// Reset FB
IF ( NOT Execute )
THEN
  Reset(); 
END_IF
END_METHOD

METHOD INTERNAL ParseResponsePayload : DINT
VAR_INPUT
  /// Response data
  ResponseData : RobotLibraryRecvDataFB;
  /// Timestamp
  Timestamp    : SystemTime;  
END_VAR
// TTable 6-172: Received CMD payload (RC to PLC) of "ReadLoadData"
// --------------------------
// Header
// --------------------------
// Byte 00 : USINT   - ParSeq | State     
// Byte 01 : SINT    - AlarmMessageSeverity    
// Byte 02 : UINT    - AlarmMessageCode HB
// Byte 03 :         - AlarmMessageCode LB
// --------------------------
// Datablock
// --------------------------
// Byte 04 : DATE    - LoadData.Date LW HB;
// Byte 05 :         - LoadData.Date LW LB;
// Byte 06 : TOD     - LoadData.Time LW HB;
// Byte 07 :         - LoadData.Time LW LB;
// Byte 08 :         - LoadData.Time LW HB;
// Byte 09 :         - LoadData.Time LW LB;
// Byte 10 : REAL    - LoadData.X HW HB;
// Byte 11 :         - LoadData.X HW LB;
// Byte 12 :         - LoadData.X LW HB;
// Byte 13 :         - LoadData.X LW LB;
// Byte 14 : REAL    - LoadData.Y HW HB;
// Byte 15 :         - LoadData.Y HW LB;
// Byte 16 :         - LoadData.Y LW HB;
// Byte 17 :         - LoadData.Y LW LB;
// Byte 18 : REAL    - LoadData.Z HW HB;
// Byte 19 :         - LoadData.Z HW LB;
// Byte 20 :         - LoadData.Z LW HB;
// Byte 21 :         - LoadData.Z LW LB;
// Byte 22 : REAL    - LoadData.RX HW HB;
// Byte 23 :         - LoadData.RX HW LB;
// Byte 24 :         - LoadData.RX LW HB;
// Byte 25 :         - LoadData.RX LW LB;
// Byte 26 : REAL    - LoadData.RY HW HB;
// Byte 27 :         - LoadData.RY HW LB;
// Byte 28 :         - LoadData.RY LW HB;
// Byte 29 :         - LoadData.RY LW LB;
// Byte 30 : REAL    - LoadData.RZ HW HB;
// Byte 31 :         - LoadData.RZ HW LB;
// Byte 32 :         - LoadData.RZ LW HB;
// Byte 33 :         - LoadData.RZ LW LB;
// Byte 34 : REAL    - LoadData.Mass HW HB;
// Byte 35 :         - LoadData.Mass HW LB;
// Byte 36 :         - LoadData.Mass LW HB;
// Byte 37 :         - LoadData.Mass LW LB;
// Byte 38 : REAL    - LoadData.IX HW HB;
// Byte 39 :         - LoadData.IX HW LB;
// Byte 40 :         - LoadData.IX LW HB;
// Byte 41 :         - LoadData.IX LW LB;
// Byte 42 : REAL    - LoadData.IY HW HB;
// Byte 43 :         - LoadData.IY HW LB;
// Byte 44 :         - LoadData.IY LW HB;
// Byte 45 :         - LoadData.IY LW LB;
// Byte 46 : REAL    - LoadData.IZ HW HB;
// Byte 47 :         - LoadData.IZ HW LB;
// Byte 48 :         - LoadData.IZ LW HB;
// Byte 49 :         - LoadData.IZ LW LB;
// Byte 50 : USINT   - LoadNo;
// Byte 51 : BOOL    - DataChanged;
// --------------------------
// call base implementation to parse the header from payload buffer
ResponseData.PayloadPtr := SUPER^.ParseResponsePayload(ResponseData := ResponseData, Timestamp := Timestamp);

// copy parsed header to response
_response.ParSeq               := _rspHeader.ParSeq;
_response.State                := _rspHeader.State;
_response.AlarmMessageSeverity := _rspHeader.AlarmMessageSeverity;
_response.AlarmMessageCode     := _rspHeader.AlarmMessageCode;

// Get Response.LoadData.Timestamp.IEC_DATE
_response.LoadData.Timestamp.IEC_DATE := ResponseData.GetIecDate();
// Get Response.LoadData.Timestamp.IEC_TIME
_response.LoadData.Timestamp.IEC_TIME := ResponseData.GetIecTime();
// Get Response.LoadData.X
_response.LoadData.X := ResponseData.GetReal();
// Get Response.LoadData.Y
_response.LoadData.Y := ResponseData.GetReal();
// Get Response.LoadData.Z
_response.LoadData.Z := ResponseData.GetReal();
// Get Response.LoadData.Rx
_response.LoadData.Rx := ResponseData.GetReal();
// Get Response.LoadData.Ry
_response.LoadData.Ry := ResponseData.GetReal();
// Get Response.LoadData.Rz
_response.LoadData.Rz := ResponseData.GetReal();
// Get Response.LoadData.Mass
_response.LoadData.Mass := ResponseData.GetReal();
// Get Response.LoadData.Ix
_response.LoadData.Ix := ResponseData.GetReal();
// Get Response.LoadData.Iy
_response.LoadData.Iy := ResponseData.GetReal();
// Get Response.LoadData.Iz
_response.LoadData.Iz := ResponseData.GetReal();
// Get Response.LoadNoReturn
_response.LoadNoReturn := ResponseData.GetUsint();
// Get Response.DataChanged
_response.DataChanged := ResponseData.GetBool();

// Create logging
ParseResponsePayloadLog(ResponseData := ResponseData, Timestamp := Timestamp);
END_METHOD

METHOD INTERNAL ParseResponsePayloadLog
VAR_INPUT
  /// Response data
  ResponseData : RobotLibraryRecvDataFB;
  /// Timestamp
  Timestamp    : SystemTime;  
END_VAR
// Create log entry for Parameter start
CreateLogMessage      ( Timestamp   := Timestamp,
                        MessageType := MessageType.CMD,
                        Severity    := Severity.DEBUG,
                        MessageCode := 0,
                        MessageText := 'Parsed the following parameter(s) from response data:');

// Create log entry for LoadData.Timestamp.IEC_DATE
CreateLogMessagePara1 ( Timestamp   := Timestamp,
                        MessageType := MessageType.CMD,
                        Severity    := Severity.DEBUG,
                        MessageCode := 0,
                        MessageText := 'Response.LoadData.Timestamp.IEC_DATE = {1}',
                        Para1       :=  IEC_DATE_TO_STRING(_response.LoadData.Timestamp.IEC_DATE));

// Create log entry for LoadData.Timestamp.IEC_TIME
CreateLogMessagePara1 ( Timestamp   := Timestamp,
                        MessageType := MessageType.CMD,
                        Severity    := Severity.DEBUG,
                        MessageCode := 0,
                        MessageText := 'Response.LoadData.Timestamp.IEC_TIME = {1}',
                        Para1       :=  IEC_TIME_TO_STRING(_response.LoadData.Timestamp.IEC_TIME));
                        
// Create log entry for LoadData.X
CreateLogMessagePara1 ( Timestamp   := Timestamp,
                        MessageType := MessageType.CMD,
                        Severity    := Severity.DEBUG,
                        MessageCode := 0,
                        MessageText := 'Response.LoadData.X = {1}',
                        Para1       :=  REAL_TO_STRING(_response.LoadData.X));

// Create log entry for LoadData.Y
CreateLogMessagePara1 ( Timestamp   := Timestamp,
                        MessageType := MessageType.CMD,
                        Severity    := Severity.DEBUG,
                        MessageCode := 0,
                        MessageText := 'Response.LoadData.Y = {1}',
                        Para1       :=  REAL_TO_STRING(_response.LoadData.Y));

// Create log entry for LoadData.Z
CreateLogMessagePara1 ( Timestamp   := Timestamp,
                        MessageType := MessageType.CMD,
                        Severity    := Severity.DEBUG,
                        MessageCode := 0,
                        MessageText := 'Response.LoadData.Z = {1}',
                        Para1       :=  REAL_TO_STRING(_response.LoadData.Z));

// Create log entry for LoadData.Rx
CreateLogMessagePara1 ( Timestamp   := Timestamp,
                        MessageType := MessageType.CMD,
                        Severity    := Severity.DEBUG,
                        MessageCode := 0,
                        MessageText := 'Response.LoadData.Rx = {1}',
                        Para1       :=  REAL_TO_STRING(_response.LoadData.Rx));

// Create log entry for LoadData.Ry
CreateLogMessagePara1 ( Timestamp   := Timestamp,
                        MessageType := MessageType.CMD,
                        Severity    := Severity.DEBUG,
                        MessageCode := 0,
                        MessageText := 'Response.LoadData.Ry = {1}',
                        Para1       :=  REAL_TO_STRING(_response.LoadData.Ry));

// Create log entry for LoadData.Rz
CreateLogMessagePara1 ( Timestamp   := Timestamp,
                        MessageType := MessageType.CMD,
                        Severity    := Severity.DEBUG,
                        MessageCode := 0,
                        MessageText := 'Response.LoadData.Rz = {1}',
                        Para1       :=  REAL_TO_STRING(_response.LoadData.Rz));

// Create log entry for LoadData.Mass
CreateLogMessagePara1 ( Timestamp   := Timestamp,
                        MessageType := MessageType.CMD,
                        Severity    := Severity.DEBUG,
                        MessageCode := 0,
                        MessageText := 'Response.LoadData.Mass = {1}',
                        Para1       :=  REAL_TO_STRING(_response.LoadData.Mass));

// Create log entry for LoadData.Ix
CreateLogMessagePara1 ( Timestamp   := Timestamp,
                        MessageType := MessageType.CMD,
                        Severity    := Severity.DEBUG,
                        MessageCode := 0,
                        MessageText := 'Response.LoadData.Ix = {1}',
                        Para1       :=  REAL_TO_STRING(_response.LoadData.Ix));

// Create log entry for LoadData.Iz
CreateLogMessagePara1 ( Timestamp   := Timestamp,
                        MessageType := MessageType.CMD,
                        Severity    := Severity.DEBUG,
                        MessageCode := 0,
                        MessageText := 'Response.LoadData.Iz = {1}',
                        Para1       :=  REAL_TO_STRING(_response.LoadData.Iz));

// Create log entry for LoadData.Iy
CreateLogMessagePara1 ( Timestamp   := Timestamp,
                        MessageType := MessageType.CMD,
                        Severity    := Severity.DEBUG,
                        MessageCode := 0,
                        MessageText := 'Response.LoadData.Iy = {1}',
                        Para1       :=  REAL_TO_STRING(_response.LoadData.Iy));

  // Create log entry for LoadNoReturn
CreateLogMessagePara1 ( Timestamp   := Timestamp,
                        MessageType := MessageType.CMD,
                        Severity    := Severity.DEBUG,
                        MessageCode := 0,
                        MessageText := 'Response.LoadNoReturn = {1}',
                        Para1       :=  USINT_TO_STRING(_response.LoadNoReturn));

  // Create log entry for DataChanged
CreateLogMessagePara1 ( Timestamp   := Timestamp,
                        MessageType := MessageType.CMD,
                        Severity    := Severity.DEBUG,
                        MessageCode := 0,
                        MessageText := 'Response.DataChanged = {1}',
                        Para1       :=  BOOL_TO_STRING(_response.DataChanged));
END_METHOD

METHOD PROTECTED Reset : DINT
VAR_INPUT
END_VAR
Reset := SUPER^.Reset();

Done               := FALSE;
Busy               := FALSE;
CommandBuffered    := FALSE;
END_METHOD

END_FUNCTION_BLOCK

// Library/POUs/Read/MC_ReadReals/MC_ReadRealsFB
/// Read real values on RC
FUNCTION_BLOCK MC_ReadRealsFB EXTENDS RobotLibraryBaseExecuteFB
// ------------------------------------------------------------------------- 
//  SRCI Robot Library                                                
// ------------------------------------------------------------------------- 
//                                                                           
//  Object:      ReadRealsFB                                       
//  Author:      Thorsten Brach                                                
//  Date:        2024-06-01
//
//  Description:                                              
//   
//                                                                           
//  Copyright: 
//    (C) 2024 Thorsten Brach. All rights reserved                                                                                                                                            
//             Licensed under the LGPL-3.0 license.
//                                                                           
//  Disclaimer:                                                                           
//    This project is provided without any guarantee and can be used for   
//    private and commercial purposes. Any use is at the user’s 
//    own risk and responsibility.
//
// -------------------------------------------------------------------------
VAR_INPUT
  /// Processing Mode
  ProcessingMode     : ProcessingMode;
  /// Defines the target sequence in which the command will be executed
  SequenceFlag       : SequenceFlag;
  /// command parameter 
  ParCmd             : ReadRealsParCmd;
END_VAR
VAR_OUTPUT
  /// TRUE, while the following outputs return valid values:
  /// • Values
  Valid              : BOOL; 
  /// Command is transferred and confirmed by the RC
  CommandBuffered    : BOOL;
  /// The command was aborted by another command.
  CommandAborted     : BOOL;
  /// TRUE, while command is interrupted during execution and can be continued
  CommandInterrupted : BOOL;
  /// command outputs
  OutCmd             : ReadRealsOutCmd;       
END_VAR

VAR
  /// internal copy of command parameter 
 _parCmd             : ReadRealsParCmd;
  /// command data to send
 _command            : ReadRealsSendData;
  /// response data received
 _response           : ReadRealsRecvData;      
END_VAR

SUPER^(AxesGroup := AxesGroup);

METHOD PROTECTED CheckFunctionSupported : BOOL
VAR_IN_OUT
  /// Robot assignment of function
  AxesGroup : AxesGroup; 
END_VAR
CheckFunctionSupported := AxesGroup.InternalData.RCSupportedFunctions.ReadReals;

IF ( NOT CheckFunctionSupported )
THEN
  // call base implementation for set error and create log entry
  SUPER^.CheckFunctionSupported(AxesGroup := AxesGroup);
END_IF
END_METHOD

METHOD PROTECTED CheckParameterChanged : BOOL
VAR_IN_OUT
  /// Robot assignment of function
  AxesGroup    : AxesGroup; 
END_VAR
// Check ParCmd Size is > 0, because MemCmp does not work correctly with size = 0
IF (SIZEOF(ParCmd) = 0) 
THEN 
  RETURN;
END_IF

// compare memory 
_parameterChanged := ( SysDepMemCmp(pData1 := ADR(ParCmd), pData2 := ADR(_parCmd), DataLen := SIZEOF(ParCmd)) <> RobotLibraryConstants.OK );

// check parameter valid ?
_parameterValid   := CheckParameterValid( AxesGroup := AxesGroup );

IF ((  _parameterChanged        )  AND 
    (  _parameterValid          )) OR
    (  _parameterUpdateInternal )  
THEN  
  // reset internal flag for send parameter update
 _parameterUpdateInternal := FALSE;
  // update internal copy of parameters 
 _parCmd := ParCmd;
  // inc parameter sequence
 _command.ParSeq := _command.ParSeq + 1;
  // update command data  
  CommandData := CreateCommandPayload(AxesGroup := AxesGroup); // ( Access via reference to rCommandFB in ACR )
  // notify active command register 
  AxesGroup.Acyclic.ActiveCommandRegister.NotifyParameterChanged := _uniqueID;
END_IF
END_METHOD

METHOD INTERNAL CreateCommandPayload : RobotLibrarySendDataFB
VAR_IN_OUT
  /// Robot assignment of function
  AxesGroup : AxesGroup; 
END_VAR
// Table 6-502: Sent CMD payload (PLC to RC) of "ReadReals"
// --------------------------
// Header
// --------------------------
// Byte 00 : UINT  - Type HB     
// Byte 01 :       - Type LB    
// Byte 02 : USINT - Reserve | ExecutionMode
// Byte 03 : USINT - ParSeq  | Priority
// --------------------------
// Datablock
// --------------------------
// Byte 04 : SINT  EmitterID[0];
// Byte 05 : SINT  EmitterID[1];
// Byte 06 : SINT  EmitterID[2];
// Byte 07 : SINT  EmitterID[3];
// Byte 08 : SINT  ListenerID;
// Byte 09 : BYTE  Reserved;
// Byte 10 : USINT Index[0];
// Byte 11 : USINT Index[1];
// Byte 12 : USINT Index[2];
// Byte 13 : USINT Index[3];
// Byte 14 : USINT Index[4];
// Byte 14 : USINT Index[5];
// Byte 14 : USINT Index[6];
// --------------------------
// set command parameter 
_command.CmdTyp       :=  CmdType.ReadReals;
_command.ExecMode     :=  ExecMode;
_command.ParSeq       := _command.ParSeq;
_command.Priority     :=  Priority;
_command.EmitterID[0] := 0;
_command.EmitterID[1] := 0;
_command.EmitterID[2] := 0;
_command.EmitterID[3] := 0;
_command.Reserve      := 0;
_command.ListenerID   := _parCmd.ListenerID;
_command.Index        := _parCmd.Index;


// copy command data to header
_cmdHeader := _command;
// call base implementation to copy header to payload buffer
CreateCommandPayload := SUPER^.CreateCommandPayload(AxesGroup := AxesGroup);

// add command.EmitterID[0]
CreateCommandPayload.AddSint(_command.EmitterID[0]);
// add command.EmitterID[1]
CreateCommandPayload.AddSint(_command.EmitterID[1]);
// add command.EmitterID[2]
CreateCommandPayload.AddSint(_command.EmitterID[2]);
// add command.EmitterID[3]
CreateCommandPayload.AddSint(_command.EmitterID[3]);
// add command.ListenerID
CreateCommandPayload.AddSint(_command.ListenerID);
// add command.Reserve
CreateCommandPayload.AddSint(_command.Reserve);
// add command.Index[0]
CreateCommandPayload.AddUsint(_command.Index[0]);
// add command.Index[1]
CreateCommandPayload.AddUsint(_command.Index[1]);
// add command.Index[2]
CreateCommandPayload.AddUsint(_command.Index[2]);
// add command.Index[3]
CreateCommandPayload.AddUsint(_command.Index[3]);
// add command.Index[4]
CreateCommandPayload.AddUsint(_command.Index[4]);
// add command.Index[5]
CreateCommandPayload.AddUsint(_command.Index[5]);
// add command.Index[6]
CreateCommandPayload.AddUsint(_command.Index[6]);

// Create logging
CreateCommandPayloadLog(AxesGroup := AxesGroup);
END_METHOD

METHOD INTERNAL CreateCommandPayloadLog
VAR_IN_OUT
  /// Robot assignment of function
  AxesGroup : AxesGroup; 
END_VAR
VAR 
  /// internal index for loops
 _idx : DINT;
END_VAR
// Create log entry for Parameter start
CreateLogMessage      ( Timestamp   := AxesGroup.InternalData.SystemTime,
                        MessageType := MessageType.CMD,
                        Severity    := Severity.DEBUG,
                        MessageCode := 0,
                        MessageText := 'Create command payload with the following parameter(s) :');
  
// Create log entry for EmitterID[x]
FOR _idx := 0 TO 3
DO
  CreateLogMessagePara2 ( Timestamp   := AxesGroup.InternalData.SystemTime,
                          MessageType := MessageType.CMD,
                          Severity    := Severity.DEBUG,
                          MessageCode := 0,
                          MessageText := 'Command.EmitterID[{2}] = {1}',
                          Para1       :=  SINT_TO_STRING(_command.EmitterID[_idx]),
                          Para2       :=  DINT_TO_STRING(_idx));
END_FOR

// Create log entry for ListenerID
CreateLogMessagePara1 ( Timestamp   := AxesGroup.InternalData.SystemTime,
                        MessageType := MessageType.CMD,
                        Severity    := Severity.DEBUG,
                        MessageCode := 0,
                        MessageText := 'Command.ListenerID = {1}',
                        Para1       :=  SINT_TO_STRING(_command.ListenerID));
                        
// Create log entry for Reserve
CreateLogMessagePara1 ( Timestamp   := AxesGroup.InternalData.SystemTime,
                        MessageType := MessageType.CMD,
                        Severity    := Severity.DEBUG,
                        MessageCode := 0,
                        MessageText := 'Command.Reserve = {1}',
                        Para1       :=  SINT_TO_STRING(_command.Reserve));

// Create log entry for Index[x]
FOR _idx := 0 TO 6
DO
  CreateLogMessagePara2 ( Timestamp   := AxesGroup.InternalData.SystemTime,
                          MessageType := MessageType.CMD,
                          Severity    := Severity.DEBUG,
                          MessageCode := 0,
                          MessageText := 'Command.Index[{2}] = {1}',
                          Para1       :=  USINT_TO_STRING(_command.Index[_idx]),
                          Para2       :=  DINT_TO_STRING(_idx));
END_FOR
END_METHOD

METHOD FB_init : BOOL
VAR_INPUT
  /// if TRUE, the retain variables are initialized (warm start / cold start)
  bInitRetains : BOOL; 
  /// if TRUE, the instance afterwards gets moved into the copy code (online change)
  bInCopyCode  : BOOL;  
END_VAR
MyType := 'MC_ReadRealsFB';

ExecMode := ExecutionMode.PARALLEL;
END_METHOD

METHOD PROTECTED OnCall
VAR_IN_OUT
  /// Robot assignment of function
  AxesGroup : AxesGroup; 
END_VAR
// call base implementation
SUPER^.OnCall(AxesGroup := AxesGroup);

CASE _stepCmd OF
  
  00:  IF ( _execute_R.Q )  
       THEN
         // Check function is supported and parameter are valid ?
         IF (( CheckFunctionSupported( AxesGroup := AxesGroup )) AND
             ( CheckParameterValid   ( AxesGroup := AxesGroup )))
         THEN      
           // set busy flag
           Busy := TRUE;
           // Reset command outputs
           SysDepMemSet(pDest := ADR(OutCmd), Value := 0, DataLen := SIZEOF(OutCmd));         
           // apply command parameter
          _parCmd := ParCmd;
           // init parameter sequence
          _command.ParSeq := 1;
           // create command data
           CommandData := CreateCommandPayload(AxesGroup := AxesGroup);
           // Add command to active command register
          _uniqueID := AxesGroup.Acyclic.ActiveCommandRegister.AddCmd( pCommandFB := ADR(THIS^ ));     
           // set timeout
           SetTimeout(PT := _timeoutCmd, rTimer := _timerCmd);
           // inc step counter
          _stepCmd := _stepCmd + 1;
         END_IF 
       END_IF
     

  01:  // Wait for responce received
       IF ( _responseReceived )
       THEN
         // reset response received flag
        _responseReceived := FALSE;

         CASE  _response.State 
         OF
           CmdMessageState.BUFFERED    : CommandBuffered    := TRUE;
           CmdMessageState.INTERRUPTED : CommandInterrupted := TRUE;           
           CmdMessageState.DONE        : Done               := TRUE;           
           CmdMessageState.ABORTED     : CommandAborted     := TRUE;
           CmdMessageState.ERROR       : Error              := TRUE;
         END_CASE
                
         // Done, Aborted or Error ?
         IF (_response.State >= CmdMessageState.DONE )
         THEN
           // Reset Busy flag
           Busy := FALSE;
           // Update results
           OutCmd.OriginID          := _response.OriginID;
           OutCmd.InvocationCounter := _response.InvocationCounter;
           OutCmd.Values            := _response.Values;
           
           // set timeout
           SetTimeout(PT := _timeoutCmd, rTimer := _timerCmd);
           // inc step counter
          _stepCmd := _stepCmd + 1; 
         END_IF
       END_IF


  02: IF ( NOT Execute)
      THEN
        Reset();
      END_IF
     
ELSE
  // invalid step
  ErrorID := RobotLibraryEvents.ERR_INVALID_STEP;
END_CASE


// Reset FB
IF ( NOT Execute )
THEN
  Reset();
END_IF
END_METHOD

METHOD INTERNAL ParseResponsePayload : DINT
VAR_INPUT
  /// Response data
  ResponseData : RobotLibraryRecvDataFB;
  /// Timestamp
  Timestamp    : SystemTime;  
END_VAR
VAR 
  /// internal index for loops
 _idx : DINT;
END_VAR
// Table Table 6-503: Received CMD payload (RC to PLC) of "ReadReals"
// --------------------------
// Header
// --------------------------
// Byte 00 : USINT   - ParSeq | State     
// Byte 01 : SINT    - AlarmMessageSeverity    
// Byte 02 : UINT    - AlarmMessageCode HB
// Byte 03 :         - AlarmMessageCode LB
// --------------------------
// Datablock
// --------------------------
// Byte 04 : USINT   - InvocationCounter;
// Byte 05 : SINT    - Reserved;
// Byte 06 : INT     - OriginID HW HB;
// Byte 07 :         - OriginID HW LB;
// Byte 08 : REAL    - Values[0] HW HB;
// Byte 09 :         - Values[0] HW LB;
// Byte 10 :         - Values[0] LW HB;
// Byte 11 :         - Values[0] LW LB;
// Byte 12 : REAL    - Values[1] HW HB;
// Byte 13 :         - Values[1] HW LB;
// Byte 14 :         - Values[1] LW HB;
// Byte 15 :         - Values[1] LW LB;
// Byte 16 : REAL    - Values[2] HW HB;
// Byte 17 :         - Values[2] HW LB;
// Byte 18 :         - Values[2] LW HB;
// Byte 19 :         - Values[2] LW LB;
// Byte 20 : REAL    - Values[3] HW HB;
// Byte 21 :         - Values[3] HW LB;
// Byte 22 :         - Values[3] LW HB;
// Byte 23 :         - Values[3] LW LB;
// Byte 24 : REAL    - Values[4] HW HB;
// Byte 25 :         - Values[4] HW LB;
// Byte 26 :         - Values[4] LW HB;
// Byte 27 :         - Values[4] LW LB;
// Byte 28 : REAL    - Values[5] HW HB;
// Byte 29 :         - Values[5] HW LB;
// Byte 30 :         - Values[5] LW HB;
// Byte 31 :         - Values[5] LW LB;
// Byte 32 : REAL    - Values[6] HW HB;
// Byte 33 :         - Values[6] HW LB;
// Byte 34 :         - Values[6] LW HB;
// Byte 35 :         - Values[6] LW LB;
// --------------------------
// call base implementation to parse the header from payload buffer
ResponseData.PayloadPtr := SUPER^.ParseResponsePayload(ResponseData := ResponseData, Timestamp := Timestamp);

// copy parsed header to response
_response.ParSeq               := _rspHeader.ParSeq;
_response.State                := _rspHeader.State;
_response.AlarmMessageSeverity := _rspHeader.AlarmMessageSeverity;
_response.AlarmMessageCode     := _rspHeader.AlarmMessageCode;

// Get Response.InvocationCounter
_response.InvocationCounter := ResponseData.GetUsint();
// Get Response.Reserve
_response.Reserve := ResponseData.GetSint();
// Get Response.OriginID/
_response.OriginID := ResponseData.GetInt();

// Get Response.Values[0]
FOR _idx := 0 TO 6 
DO
 _response.Values[_idx] := ResponseData.GetReal();
END_FOR

// Create logging
ParseResponsePayloadLog(ResponseData := ResponseData, Timestamp := Timestamp);
END_METHOD

METHOD INTERNAL ParseResponsePayloadLog
VAR_INPUT
  /// Response data
  ResponseData : RobotLibraryRecvDataFB;
  /// Timestamp
  Timestamp    : SystemTime;  
END_VAR
VAR 
  /// internal index for loops
 _idx : DINT;
END_VAR
// Create log entry for Parameter start
CreateLogMessage      ( Timestamp   := Timestamp,
                        MessageType := MessageType.CMD,
                        Severity    := Severity.DEBUG,
                        MessageCode := 0,
                        MessageText := 'Parsed the following parameter(s) from response data:');
                        
// Create log entry for InvocationCounter
CreateLogMessagePara1 ( Timestamp   := Timestamp,
                        MessageType := MessageType.CMD,
                        Severity    := Severity.DEBUG,
                        MessageCode := 0,
                        MessageText := 'Response.InvocationCounter = {1}',
                        Para1       :=  USINT_TO_STRING(_response.InvocationCounter));

// Create log entry for Reserve
CreateLogMessagePara1 ( Timestamp   := Timestamp,
                        MessageType := MessageType.CMD,
                        Severity    := Severity.DEBUG,
                        MessageCode := 0,
                        MessageText := 'Response.Reserve = {1}',
                        Para1       :=  SINT_TO_STRING(_response.Reserve));

// Create log entry for OriginID
CreateLogMessagePara1 ( Timestamp   := Timestamp,
                        MessageType := MessageType.CMD,
                        Severity    := Severity.DEBUG,
                        MessageCode := 0,
                        MessageText := 'Response.OriginID = {1}',
                        Para1       :=  INT_TO_STRING(_response.OriginID));

// Create log entry for Values[{x}]
FOR _idx := 0 TO 6
DO
  CreateLogMessagePara2 ( Timestamp   := Timestamp,
                          MessageType := MessageType.CMD,
                          Severity    := Severity.DEBUG,
                          MessageCode := 0,
                          MessageText := 'Response.Values[{2}] = {1}',
                          Para1       :=  REAL_TO_STRING(_response.Values[_idx]),
                          Para2       :=  DINT_TO_STRING(_idx));
END_FOR
END_METHOD

METHOD PROTECTED Reset : DINT
VAR_INPUT
END_VAR
Reset := SUPER^.Reset();

Done               := FALSE;
Busy               := FALSE;
Valid              := FALSE; 
CommandBuffered    := FALSE;
CommandAborted     := FALSE;
CommandInterrupted := FALSE;
END_METHOD

END_FUNCTION_BLOCK

// Library/POUs/Read/MC_ReadRobotDefaultDynamics/MC_ReadRobotDefaultDynamicsFB
/// Read default values of dynamic parameters used by move commands
FUNCTION_BLOCK MC_ReadRobotDefaultDynamicsFB EXTENDS RobotLibraryBaseExecuteFB
// ------------------------------------------------------------------------- 
//  SRCI Robot Library                                                
// ------------------------------------------------------------------------- 
//                                                                           
//  Object:      ReadRobotDefaultDynamicsFB                                       
//  Author:      Thorsten Brach                                                
//  Date:        2024-06-01
//
//  Description:                                              
//   
//                                                                           
//  Copyright: 
//    (C) 2024 Thorsten Brach. All rights reserved                                                                                                                                            
//             Licensed under the LGPL-3.0 license.
//                                                                           
//  Disclaimer:                                                                           
//    This project is provided without any guarantee and can be used for   
//    private and commercial purposes. Any use is at the user’s 
//    own risk and responsibility.
//
// -------------------------------------------------------------------------
VAR_INPUT
  /// command parameter 
  ParCmd          : ReadRobotDefaultDynamicsParCmd;  
END_VAR

VAR_OUTPUT
  /// Command is transferred and confirmed by the RC
  CommandBuffered : BOOL;
  /// command outputs
  OutCmd          : ReadRobotDefaultDynamicsOutCmd;       
END_VAR

VAR
  /// internal copy of command parameter 
 _parCmd          : ReadRobotDefaultDynamicsParCmd;
  /// command data to send
 _command         : ReadRobotDefaultDynamicsSendData;
  /// response data received
 _response        : ReadRobotDefaultDynamicsRecvData;      
END_VAR

SUPER^(AxesGroup := AxesGroup);

METHOD PROTECTED CheckFunctionSupported : BOOL
VAR_IN_OUT
  /// Robot assignment of function
  AxesGroup : AxesGroup; 
END_VAR
CheckFunctionSupported := AxesGroup.InternalData.RCSupportedFunctions.ReadRobotDefaultDynamics;

IF ( NOT CheckFunctionSupported )
THEN
  // call base implementation for set error and create log entry
  SUPER^.CheckFunctionSupported(AxesGroup := AxesGroup);
END_IF
END_METHOD

METHOD PROTECTED CheckParameterChanged : BOOL
VAR_IN_OUT
  /// Robot assignment of function
  AxesGroup    : AxesGroup; 
END_VAR
// Check ParCmd Size is > 0, because MemCmp does not work correctly with size = 0
IF (SIZEOF(ParCmd) = 0) 
THEN 
  RETURN;
END_IF

// compare memory 
_parameterChanged := ( SysDepMemCmp(pData1 := ADR(ParCmd), pData2 := ADR(_parCmd), DataLen := SIZEOF(ParCmd)) <> RobotLibraryConstants.OK );

// check parameter valid ?
_parameterValid   := CheckParameterValid( AxesGroup := AxesGroup );

IF ((  _parameterChanged        )  AND 
    (  _parameterValid          )) OR
    (  _parameterUpdateInternal )  
THEN  
  // reset internal flag for send parameter update
 _parameterUpdateInternal := FALSE;
  // update internal copy of parameters 
 _parCmd := ParCmd;
  // inc parameter sequence
 _command.ParSeq := _command.ParSeq + 1;
  // update command data  
  CommandData := CreateCommandPayload(AxesGroup := AxesGroup); // ( Access via reference to rCommandFB in ACR )
  // notify active command register 
  AxesGroup.Acyclic.ActiveCommandRegister.NotifyParameterChanged := _uniqueID;
END_IF
END_METHOD

METHOD INTERNAL CreateCommandPayload : RobotLibrarySendDataFB
VAR_IN_OUT
  /// Robot assignment of function
  AxesGroup : AxesGroup; 
END_VAR
// Table 6-153: Sent CMD payload (PLC to RC) of "ReadRobotDefaultDynamics"
// --------------------------
// Header
// --------------------------
// Byte 00 : UINT  - Type HB     
// Byte 01 :       - Type LB    
// Byte 02 : USINT - Reserve | ExecutionMode
// Byte 03 : USINT - ParSeq  | Priority
// --------------------------
// set command parameter 
_command.CmdTyp   :=  CmdType.ReadRobotDefaultDynamics;
_command.ExecMode :=  ExecMode;
_command.ParSeq   := _command.ParSeq;
_command.Priority :=  Priority;

// copy command data to header
_cmdHeader := _command;
// call base implementation to copy header to payload buffer
CreateCommandPayload := SUPER^.CreateCommandPayload(AxesGroup := AxesGroup);

// Create logging
CreateCommandPayloadLog(AxesGroup := AxesGroup);
END_METHOD

METHOD INTERNAL CreateCommandPayloadLog
VAR_IN_OUT
  /// Robot assignment of function
  AxesGroup : AxesGroup; 
END_VAR
// Create log entry for Parameter start
CreateLogMessage      ( Timestamp   := AxesGroup.InternalData.SystemTime,
                        MessageType := MessageType.CMD,
                        Severity    := Severity.DEBUG,
                        MessageCode := 0,
                        MessageText := 'Create command payload without additional parameter(s)');
END_METHOD

METHOD FB_init : BOOL
VAR_INPUT
  /// if TRUE, the retain variables are initialized (warm start / cold start)
  bInitRetains : BOOL; 
  /// if TRUE, the instance afterwards gets moved into the copy code (online change)
  bInCopyCode  : BOOL;  
END_VAR
MyType := 'MC_ReadRobotDefaultDynamicsFB';

ExecMode := ExecutionMode.PARALLEL;
END_METHOD

METHOD PROTECTED OnCall
VAR_IN_OUT
  /// Robot assignment of function
  AxesGroup : AxesGroup; 
END_VAR
// call base implementation
SUPER^.OnCall(AxesGroup := AxesGroup);

CASE _stepCmd OF
  
  00:  IF ( _execute_R.Q ) 
       THEN
         // Check function is supported and parameter are valid ?
         IF (( CheckFunctionSupported( AxesGroup := AxesGroup )) AND
             ( CheckParameterValid   ( AxesGroup := AxesGroup )))
         THEN      
           // set busy flag
           Busy := TRUE;
           // Reset command outputs
           SysDepMemSet(pDest := ADR(OutCmd), Value := 0, DataLen := SIZEOF(OutCmd));         
           // apply command parameter
          _parCmd := ParCmd;
           // init parameter sequence
          _command.ParSeq := 1;
           // create command data
           CommandData := CreateCommandPayload(AxesGroup := AxesGroup);
           // Add command to active command register
          _uniqueID := AxesGroup.Acyclic.ActiveCommandRegister.AddCmd( pCommandFB := ADR(THIS^ ));     
           // set timeout
           SetTimeout(PT := _timeoutCmd, rTimer := _timerCmd);
           // inc step counter
          _stepCmd := _stepCmd + 1;
         END_IF 
       END_IF
     

  01:  // Wait for responce received
       IF ( _responseReceived )
       THEN
         // reset response received flag
        _responseReceived := FALSE;

         CASE  _response.State 
         OF
           CmdMessageState.BUFFERED : CommandBuffered := TRUE;
           CmdMessageState.DONE     : Done            := TRUE;
           CmdMessageState.ERROR    : Error           := TRUE;
         END_CASE
                
         // Done, Aborted or Error ?
         IF (_response.State >= CmdMessageState.DONE )
         THEN
           // Reset Busy flag
           Busy := FALSE;
           // Update results
           OutCmd.DynamicValues.Timestamp        := _response.Timestamp;
           OutCmd.DynamicValues.VelocityRate     :=  PERCENT_INT_TO_REAL(UINT_TO_INT(_response.VelocityRate    ), IsOptional := FALSE);
           OutCmd.DynamicValues.AccelerationRate :=  PERCENT_INT_TO_REAL(UINT_TO_INT(_response.AccelerationRate), IsOptional := FALSE);
           OutCmd.DynamicValues.DecelerationRate :=  PERCENT_INT_TO_REAL(UINT_TO_INT(_response.DecelerationRate), IsOptional := TRUE);
           OutCmd.DynamicValues.JerkRate         :=  PERCENT_INT_TO_REAL(UINT_TO_INT(_response.JerkRate        ), IsOptional := TRUE);
           
           // set timeout
           SetTimeout(PT := _timeoutCmd, rTimer := _timerCmd);
           // inc step counter
          _stepCmd := _stepCmd + 1; 
         END_IF
       END_IF


  02: IF ( NOT Execute)
      THEN
        Reset();
      END_IF     

ELSE
  // invalid step
  ErrorID := RobotLibraryEvents.ERR_INVALID_STEP;
END_CASE


// Reset FB
IF ( NOT Execute )
THEN
  Reset();
END_IF
END_METHOD

METHOD INTERNAL ParseResponsePayload : DINT
VAR_INPUT
  /// Response data
  ResponseData : RobotLibraryRecvDataFB;
  /// Timestamp
  Timestamp    : SystemTime;  
END_VAR
// Table 6-154: Received CMD payload (RC to PLC) of "ReadRobotDefaultDynamics"
// --------------------------
// Header
// --------------------------
// Byte 00 : USINT   - ParSeq | State     
// Byte 01 : SINT    - AlarmMessageSeverity    
// Byte 02 : UINT    - AlarmMessageCode HB
// Byte 03 :         - AlarmMessageCode LB
// --------------------------
// Datablock
// --------------------------
// Byte 04 : DATE        Date HW HB;
// Byte 05 :             Date HW LB;
// Byte 06 : TIME_OF_DAY Time HW HB;
// Byte 07 :             Time HW LB;
// Byte 08 :             Time LW HB;
// Byte 09 :             Time LW LB;
// Byte 10 : UINT        VelocityRate HW HB;
// Byte 11 :             VelocityRate HW LB;
// Byte 12 : UINT        AccelerationRate HW HB;
// Byte 13 :             AccelerationRate HW LB;
// Byte 14 : UINT        DecelerationRate HW HB;
// Byte 15 :             DecelerationRate HW LB;
// Byte 16 : UINT        JerkRate HW HB;
// Byte 17 :             JerkRate HW LB;
// Byte 18 : USINT       DataChanged;
// --------------------------
// call base implementation to parse the header from payload buffer
ResponseData.PayloadPtr := SUPER^.ParseResponsePayload(ResponseData := ResponseData, Timestamp := Timestamp);

// copy parsed header to response
_response.ParSeq               := _rspHeader.ParSeq;
_response.State                := _rspHeader.State;
_response.AlarmMessageSeverity := _rspHeader.AlarmMessageSeverity;
_response.AlarmMessageCode     := _rspHeader.AlarmMessageCode;

// Get Response.DynamicValues.Timestamp.IEC_DATE
_response.Timestamp.IEC_DATE := ResponseData.GetIecDate();
// Get Response.DynamicValues.Timestamp.IEC_TIME
_response.Timestamp.IEC_TIME := ResponseData.GetIecTime();
// Get Response.DynamicValues.VelocityRate
_response.VelocityRate := ResponseData.GetUint();
// Get Response.DynamicValues.AccelerationRate
_response.AccelerationRate := ResponseData.GetUint();
// Get Response.DynamicValues.DecelerationRate
_response.DecelerationRate := ResponseData.GetUint();
// Get Response.DynamicValues.JerkRate
_response.JerkRate := ResponseData.GetUint();
// Get Response.DataChanged
_response.DataChanged := ResponseData.GetBool();

// Create logging
ParseResponsePayloadLog(ResponseData := ResponseData, Timestamp := Timestamp);
END_METHOD

METHOD INTERNAL ParseResponsePayloadLog
VAR_INPUT
  /// Response data
  ResponseData : RobotLibraryRecvDataFB;
  /// Timestamp
  Timestamp    : SystemTime;  
END_VAR
// Create log entry for Parameter start
CreateLogMessage      ( Timestamp   := Timestamp,
                        MessageType := MessageType.CMD,
                        Severity    := Severity.DEBUG,
                        MessageCode := 0,
                        MessageText := 'Parsed the following parameter(s) from response data:');
                        
// Create log entry for Timestamp.IEC_DATE
CreateLogMessagePara1 ( Timestamp   := Timestamp,
                        MessageType := MessageType.CMD,
                        Severity    := Severity.DEBUG,
                        MessageCode := 0,
                        MessageText := 'Response.Timestamp.IEC_DATE = {1}',
                        Para1       :=  IEC_DATE_TO_STRING(_response.Timestamp.IEC_DATE));

// Create log entry for Timestamp.IEC_TIME
CreateLogMessagePara1 ( Timestamp   := Timestamp,
                        MessageType := MessageType.CMD,
                        Severity    := Severity.DEBUG,
                        MessageCode := 0,
                        MessageText := 'Response.Timestamp.IEC_TIME = {1}',
                        Para1       :=  IEC_TIME_TO_STRING(_response.Timestamp.IEC_TIME));
                        
// Create log entry for VelocityRate
CreateLogMessagePara1 ( Timestamp   := Timestamp,
                        MessageType := MessageType.CMD,
                        Severity    := Severity.DEBUG,
                        MessageCode := 0,
                        MessageText := 'Response.VelocityRate = {1}',
                        Para1       :=  UINT_TO_STRING(_response.VelocityRate));

// Create log entry for AccelerationRate
CreateLogMessagePara1 ( Timestamp   := Timestamp,
                        MessageType := MessageType.CMD,
                        Severity    := Severity.DEBUG,
                        MessageCode := 0,
                        MessageText := 'Response.AccelerationRate = {1}',
                        Para1       :=  UINT_TO_STRING(_response.AccelerationRate));

// Create log entry for DecelerationRate
CreateLogMessagePara1 ( Timestamp   := Timestamp,
                        MessageType := MessageType.CMD,
                        Severity    := Severity.DEBUG,
                        MessageCode := 0,
                        MessageText := 'Response.DecelerationRate = {1}',
                        Para1       :=  UINT_TO_STRING(_response.DecelerationRate));

// Create log entry for JerkRate
CreateLogMessagePara1 ( Timestamp   := Timestamp,
                        MessageType := MessageType.CMD,
                        Severity    := Severity.DEBUG,
                        MessageCode := 0,
                        MessageText := 'Response.JerkRate = {1}',
                        Para1       :=  UINT_TO_STRING(_response.JerkRate));

// Create log entry for DataChanged
CreateLogMessagePara1 ( Timestamp   := Timestamp,
                        MessageType := MessageType.CMD,
                        Severity    := Severity.DEBUG,
                        MessageCode := 0,
                        MessageText := 'Response.DataChanged = {1}',
                        Para1       :=  BOOL_TO_STRING(_response.DataChanged));
END_METHOD

METHOD PROTECTED Reset : DINT
VAR_INPUT
END_VAR
Reset := SUPER^.Reset();

Done               := FALSE;
Busy               := FALSE;
CommandBuffered    := FALSE;
END_METHOD

END_FUNCTION_BLOCK

// Library/POUs/Read/MC_ReadRobotReferenceDynamics/MC_ReadRobotReferenceDynamicsFB
/// Read reference values of robot dynamics for path movement
FUNCTION_BLOCK MC_ReadRobotReferenceDynamicsFB EXTENDS RobotLibraryBaseExecuteFB
// ------------------------------------------------------------------------- 
//  SRCI Robot Library                                                
// ------------------------------------------------------------------------- 
//                                                                           
//  Object:      ReadRobotReferenceDynamicsFB                                       
//  Author:      Thorsten Brach                                                
//  Date:        2024-06-01
//
//  Description:                                              
//   
//                                                                           
//  Copyright: 
//    (C) 2024 Thorsten Brach. All rights reserved                                                                                                                                            
//             Licensed under the LGPL-3.0 license.
//                                                                           
//  Disclaimer:                                                                           
//    This project is provided without any guarantee and can be used for   
//    private and commercial purposes. Any use is at the user’s 
//    own risk and responsibility.
//
// -------------------------------------------------------------------------
VAR_INPUT
  /// command parameter
  ParCmd          : ReadRobotReferenceDynamicsParCmd;       
END_VAR

VAR_OUTPUT
  /// Command is transferred and confirmed by the RC
  CommandBuffered : BOOL;
  /// command outputs
  OutCmd          : ReadRobotReferenceDynamicsOutCmd;       
END_VAR

VAR
  /// internal copy of command parameter 
 _parCmd             : ReadRobotReferenceDynamicsParCmd;
  /// command data to send
 _command            : ReadRobotReferenceDynamicsSendData;
  /// response data received
 _response           : ReadRobotReferenceDynamicsRecvData;      
END_VAR

SUPER^(AxesGroup := AxesGroup);

METHOD PROTECTED CheckFunctionSupported : BOOL
VAR_IN_OUT
  /// Robot assignment of function
  AxesGroup : AxesGroup; 
END_VAR
CheckFunctionSupported := AxesGroup.InternalData.RCSupportedFunctions.ReadRobotReferenceDynamics;

IF ( NOT CheckFunctionSupported )
THEN
  // call base implementation for set error and create log entry
  SUPER^.CheckFunctionSupported(AxesGroup := AxesGroup);
END_IF
END_METHOD

METHOD PROTECTED CheckParameterChanged : BOOL
VAR_IN_OUT
  /// Robot assignment of function
  AxesGroup    : AxesGroup; 
END_VAR
// Check ParCmd Size is > 0, because MemCmp does not work correctly with size = 0
IF (SIZEOF(ParCmd) = 0) 
THEN 
  RETURN;
END_IF

// compare memory 
_parameterChanged := ( SysDepMemCmp(pData1 := ADR(ParCmd), pData2 := ADR(_parCmd), DataLen := SIZEOF(ParCmd)) <> RobotLibraryConstants.OK );

// check parameter valid ?
_parameterValid   := CheckParameterValid( AxesGroup := AxesGroup );

IF ((  _parameterChanged        )  AND 
    (  _parameterValid          )) OR
    (  _parameterUpdateInternal )  
THEN  
  // reset internal flag for send parameter update
 _parameterUpdateInternal := FALSE;
  // update internal copy of parameters 
 _parCmd := ParCmd;
  // inc parameter sequence
 _command.ParSeq := _command.ParSeq + 1;
  // update command data  
  CommandData := CreateCommandPayload(AxesGroup := AxesGroup); // ( Access via reference to rCommandFB in ACR )
  // notify active command register 
  AxesGroup.Acyclic.ActiveCommandRegister.NotifyParameterChanged := _uniqueID;
END_IF
END_METHOD

METHOD INTERNAL CreateCommandPayload : RobotLibrarySendDataFB
VAR_IN_OUT
  /// Robot assignment of function
  AxesGroup : AxesGroup; 
END_VAR
// Table 6-114: Sent CMD payload (PLC to RC) of "ReadRobotReferenceDynamics"
// --------------------------
// Header
// --------------------------
// Byte 00 : UINT  - Type HB     
// Byte 01 :       - Type LB    
// Byte 02 : USINT - Reserve | ExecutionMode
// Byte 03 : USINT - ParSeq  | Priority
// set command parameter 
_command.CmdTyp   :=  CmdType.ReadRobotReferenceDynamics;
_command.ExecMode :=  ExecMode;
_command.ParSeq   := _command.ParSeq;
_command.Priority :=  Priority;

// copy command data to header
_cmdHeader := _command;
// call base implementation to copy header to payload buffer
CreateCommandPayload := SUPER^.CreateCommandPayload(AxesGroup := AxesGroup);

// Create logging
CreateCommandPayloadLog(AxesGroup := AxesGroup);
END_METHOD

METHOD INTERNAL CreateCommandPayloadLog
VAR_IN_OUT
  /// Robot assignment of function
  AxesGroup : AxesGroup; 
END_VAR
// Create log entry for Parameter start
CreateLogMessage      ( Timestamp   := AxesGroup.InternalData.SystemTime,
                        MessageType := MessageType.CMD,
                        Severity    := Severity.DEBUG,
                        MessageCode := 0,
                        MessageText := 'Create command payload without additional parameter(s)');
END_METHOD

METHOD FB_init : BOOL
VAR_INPUT
  /// if TRUE, the retain variables are initialized (warm start / cold start)
  bInitRetains : BOOL; 
  /// if TRUE, the instance afterwards gets moved into the copy code (online change)
  bInCopyCode  : BOOL;  
END_VAR
MyType := 'MC_ReadRobotReferenceDynamicsFB';

ExecMode := ExecutionMode.PARALLEL;
END_METHOD

METHOD PROTECTED OnCall
VAR_IN_OUT
  /// Robot assignment of function
  AxesGroup : AxesGroup; 
END_VAR
// call base implementation
SUPER^.OnCall(AxesGroup := AxesGroup);

CASE _stepCmd OF
  
  00:  IF ( _execute_R.Q ) 
       THEN
         // Check function is supported and parameter are valid ?
         IF (( CheckFunctionSupported( AxesGroup := AxesGroup )) AND
             ( CheckParameterValid   ( AxesGroup := AxesGroup )))
         THEN      
           // set busy flag
           Busy := TRUE;
           // Reset command outputs
           SysDepMemSet(pDest := ADR(OutCmd), Value := 0, DataLen := SIZEOF(OutCmd));         
           // apply command parameter
          _parCmd := ParCmd;
           // init parameter sequence
          _command.ParSeq := 1;
           // create command data
           CommandData := CreateCommandPayload(AxesGroup := AxesGroup);
           // Add command to active command register
          _uniqueID := AxesGroup.Acyclic.ActiveCommandRegister.AddCmd( pCommandFB := ADR(THIS^ ));     
           // set timeout
           SetTimeout(PT := _timeoutCmd, rTimer := _timerCmd);
           // inc step counter
          _stepCmd := _stepCmd + 1;
         END_IF 
       END_IF
     

  01:  // Wait for responce received
       IF ( _responseReceived )
       THEN
         // reset response received flag
        _responseReceived := FALSE;

         CASE  _response.State 
         OF
           CmdMessageState.BUFFERED : CommandBuffered := TRUE;
           CmdMessageState.DONE     : Done            := TRUE;
           CmdMessageState.ERROR    : Error           := TRUE;
         END_CASE
                
         // Done, Aborted or Error ?
         IF (_response.State >= CmdMessageState.DONE )
         THEN
           // Reset Busy flag
           Busy := FALSE;
           
           // Update results
           OutCmd.DynamicValues.VelocityReference     := PERCENT_INT_TO_REAL(UINT_TO_INT(_response.VelocityReference    ), IsOptional := FALSE );
           OutCmd.DynamicValues.AccelerationReference := PERCENT_INT_TO_REAL(UINT_TO_INT(_response.AccelerationReference) ,IsOptional := FALSE);
           OutCmd.DynamicValues.DecelerationReference := PERCENT_INT_TO_REAL(UINT_TO_INT(_response.DecelerationReference), IsOptional := TRUE );
           OutCmd.DynamicValues.JerkReference         := PERCENT_INT_TO_REAL(UINT_TO_INT(_response.JerkReference        ), IsOptional := TRUE );

           // set timeout
           SetTimeout(PT := _timeoutCmd, rTimer := _timerCmd);
           // inc step counter
          _stepCmd := _stepCmd + 1; 
         END_IF
       END_IF


  02: IF ( NOT Execute)
      THEN
        Reset(); 
      END_IF     

ELSE
  // invalid step
  ErrorID := RobotLibraryEvents.ERR_INVALID_STEP;
END_CASE


// Reset FB
IF ( NOT Execute )
THEN
  Reset();
END_IF
END_METHOD

METHOD INTERNAL ParseResponsePayload : DINT
VAR_INPUT
  /// Response data
  ResponseData : RobotLibraryRecvDataFB;
  /// Timestamp
  Timestamp    : SystemTime;  
END_VAR
// Table 6-115: Received CMD payload (RC to PLC) of "ReadRobotReferenceDynamics"
// --------------------------
// Header
// --------------------------
// Byte 00 : USINT   - ParSeq | State     
// Byte 01 : SINT    - AlarmMessageSeverity    
// Byte 02 : UINT    - AlarmMessageCode HB
// Byte 03 :         - AlarmMessageCode LB
// --------------------------
// Datablock
// --------------------------
// Byte 04 : DATE        Date HW HB;
// Byte 05 :             Date HW LB;
// Byte 06 : TOD         Time HW HB;
// Byte 07 :             Time HW LB;
// Byte 08 :             Time LW HB;
// Byte 09 :             Time LW LB;
// Byte 10 : UINT        VelocityReference HW HB;
// Byte 11 :             VelocityReference HW LB;
// Byte 12 : UINT        AccelerationReference HW HB;
// Byte 13 :             AccelerationReference HW LB;
// Byte 14 : UINT        DecelerationReference HW HB;
// Byte 15 :             DecelerationReference HW LB;
// Byte 16 : UINT        JerkReference HW HB;
// Byte 17 :             JerkReference HW LB;
// Byte 18 : USINT       DataChanged;
// --------------------------
// call base implementation to parse the header from payload buffer
ResponseData.PayloadPtr := SUPER^.ParseResponsePayload(ResponseData := ResponseData, Timestamp := Timestamp);

// copy parsed header to response
_response.ParSeq               := _rspHeader.ParSeq;
_response.State                := _rspHeader.State;
_response.AlarmMessageSeverity := _rspHeader.AlarmMessageSeverity;
_response.AlarmMessageCode     := _rspHeader.AlarmMessageCode;

// Get Response.DynamicValues.Timestamp.IEC_DATE
_response.Timestamp.IEC_DATE := ResponseData.GetIecDate();
// Get Response.DynamicValues.Timestamp.IEC_TIME
_response.Timestamp.IEC_TIME := ResponseData.GetIecTime();
// Get Response.DynamicValues.VelocityRate
_response.VelocityReference := ResponseData.GetUint();
// Get Response.DynamicValues.AccelerationRate
_response.AccelerationReference := ResponseData.GetUint();
// Get Response.DynamicValues.DecelerationRate
_response.DecelerationReference := ResponseData.GetUint();
// Get Response.DynamicValues.JerkRate
_response.JerkReference := ResponseData.GetUint();
// Get Response.DataChanged
_response.DataChanged := ResponseData.GetBool();

// Create logging
ParseResponsePayloadLog(ResponseData := ResponseData, Timestamp := Timestamp);
END_METHOD

METHOD INTERNAL ParseResponsePayloadLog
VAR_INPUT
  /// Response data
  ResponseData : RobotLibraryRecvDataFB;
  /// Timestamp
  Timestamp    : SystemTime;  
END_VAR
// Create log entry for Parameter start
CreateLogMessage      ( Timestamp   := Timestamp,
                        MessageType := MessageType.CMD,
                        Severity    := Severity.DEBUG,
                        MessageCode := 0,
                        MessageText := 'Parsed the following parameter(s) from response data:');
                        
// Create log entry for Timestamp.IEC_DATE
CreateLogMessagePara1 ( Timestamp   := Timestamp,
                        MessageType := MessageType.CMD,
                        Severity    := Severity.DEBUG,
                        MessageCode := 0,
                        MessageText := 'Response.Timestamp.IEC_DATE = {1}',
                        Para1       :=  IEC_DATE_TO_STRING(_response.Timestamp.IEC_DATE));

// Create log entry for Timestamp.IEC_TIME
CreateLogMessagePara1 ( Timestamp   := Timestamp,
                        MessageType := MessageType.CMD,
                        Severity    := Severity.DEBUG,
                        MessageCode := 0,
                        MessageText := 'Response.Timestamp.IEC_TIME = {1}',
                        Para1       :=  IEC_TIME_TO_STRING(_response.Timestamp.IEC_TIME));
                        
// Create log entry for VelocityReference
CreateLogMessagePara1 ( Timestamp   := Timestamp,
                        MessageType := MessageType.CMD,
                        Severity    := Severity.DEBUG,
                        MessageCode := 0,
                        MessageText := 'Response.VelocityReference = {1}',
                        Para1       :=  UINT_TO_STRING(_response.VelocityReference));

// Create log entry for AccelerationReference
CreateLogMessagePara1 ( Timestamp   := Timestamp,
                        MessageType := MessageType.CMD,
                        Severity    := Severity.DEBUG,
                        MessageCode := 0,
                        MessageText := 'Response.AccelerationReference = {1}',
                        Para1       :=  UINT_TO_STRING(_response.AccelerationReference));

// Create log entry for DecelerationReference
CreateLogMessagePara1 ( Timestamp   := Timestamp,
                        MessageType := MessageType.CMD,
                        Severity    := Severity.DEBUG,
                        MessageCode := 0,
                        MessageText := 'Response.DecelerationReference = {1}',
                        Para1       :=  UINT_TO_STRING(_response.DecelerationReference));

// Create log entry for JerkReference
CreateLogMessagePara1 ( Timestamp   := Timestamp,
                        MessageType := MessageType.CMD,
                        Severity    := Severity.DEBUG,
                        MessageCode := 0,
                        MessageText := 'Response.JerkReference = {1}',
                        Para1       :=  UINT_TO_STRING(_response.JerkReference));

// Create log entry for DataChanged
CreateLogMessagePara1 ( Timestamp   := Timestamp,
                        MessageType := MessageType.CMD,
                        Severity    := Severity.DEBUG,
                        MessageCode := 0,
                        MessageText := 'Response.DataChanged = {1}',
                        Para1       :=  BOOL_TO_STRING(_response.DataChanged));
END_METHOD

METHOD PROTECTED Reset : DINT
VAR_INPUT
END_VAR
Reset := SUPER^.Reset();

Done               := FALSE;
Busy               := FALSE;
CommandBuffered    := FALSE;
END_METHOD

END_FUNCTION_BLOCK

// Library/POUs/Read/MC_ReadRobotSWLimits/MC_ReadRobotSWLimitsFB
/// Read actual software limits of the axes Positive and negative Limit of Joint J1…J6, E1…E6
FUNCTION_BLOCK MC_ReadRobotSWLimitsFB EXTENDS RobotLibraryBaseExecuteFB
// ------------------------------------------------------------------------- 
//  SRCI Robot Library                                                
// ------------------------------------------------------------------------- 
//                                                                           
//  Object:      ReadRobotSWLimitsFB                                       
//  Author:      Thorsten Brach                                                
//  Date:        2024-06-01
//
//  Description:                                              
//   
//                                                                           
//  Copyright: 
//    (C) 2024 Thorsten Brach. All rights reserved                                                                                                                                            
//             Licensed under the LGPL-3.0 license.
//                                                                           
//  Disclaimer:                                                                           
//    This project is provided without any guarantee and can be used for   
//    private and commercial purposes. Any use is at the user’s 
//    own risk and responsibility.
//
// -------------------------------------------------------------------------
VAR_INPUT
  /// command parameter 
  ParCmd          : ReadRobotSWLimitsParCmd;
END_VAR

VAR_OUTPUT
  /// Command is transferred and confirmed by the RC
  CommandBuffered : BOOL;
  /// command outputs
  OutCmd          : ReadRobotSWLimitsOutCmd;       
END_VAR

VAR
  /// internal copy of command parameter 
 _parCmd          : ReadRobotSWLimitsParCmd;
  /// command data to send
 _command         : ReadRobotSWLimitsSendData;
  /// response data received
 _response        : ReadRobotSWLimitsRecvData;      
END_VAR

SUPER^(AxesGroup := AxesGroup);

METHOD PROTECTED CheckFunctionSupported : BOOL
VAR_IN_OUT
  /// Robot assignment of function
  AxesGroup : AxesGroup; 
END_VAR
CheckFunctionSupported := AxesGroup.InternalData.RCSupportedFunctions.ReadRobotSWLimits;

IF ( NOT CheckFunctionSupported )
THEN
  // call base implementation for set error and create log entry
  SUPER^.CheckFunctionSupported(AxesGroup := AxesGroup);
END_IF
END_METHOD

METHOD PROTECTED CheckParameterChanged : BOOL
VAR_IN_OUT
  /// Robot assignment of function
  AxesGroup    : AxesGroup; 
END_VAR
// Check ParCmd Size is > 0, because MemCmp does not work correctly with size = 0
IF (SIZEOF(ParCmd) = 0) 
THEN 
  RETURN;
END_IF

// compare memory 
_parameterChanged := ( SysDepMemCmp(pData1 := ADR(ParCmd), pData2 := ADR(_parCmd), DataLen := SIZEOF(ParCmd)) <> RobotLibraryConstants.OK );

// check parameter valid ?
_parameterValid   := CheckParameterValid( AxesGroup := AxesGroup );

IF ((  _parameterChanged        )  AND 
    (  _parameterValid          )) OR
    (  _parameterUpdateInternal )  
THEN  
  // reset internal flag for send parameter update
 _parameterUpdateInternal := FALSE;
  // update internal copy of parameters 
 _parCmd := ParCmd;
  // inc parameter sequence
 _command.ParSeq := _command.ParSeq + 1;
  // update command data  
  CommandData := CreateCommandPayload(AxesGroup := AxesGroup); // ( Access via reference to rCommandFB in ACR )
  // notify active command register 
  AxesGroup.Acyclic.ActiveCommandRegister.NotifyParameterChanged := _uniqueID;
END_IF
END_METHOD

METHOD INTERNAL CreateCommandPayload : RobotLibrarySendDataFB
VAR_IN_OUT
  /// Robot assignment of function
  AxesGroup : AxesGroup; 
END_VAR
// Table 6-178: Sent CMD payload (PLC to RC) of "ReadRobotSWLimits"
// --------------------------
// Header
// --------------------------
// Byte 00 : UINT  - Type HB     
// Byte 01 :       - Type LB    
// Byte 02 : USINT - Reserve | ExecutionMode
// Byte 03 : USINT - ParSeq  | Priority
// set command parameter 
_command.CmdTyp   :=  CmdType.ReadRobotSWLimits;
_command.ExecMode :=  ExecMode;
_command.ParSeq   := _command.ParSeq;
_command.Priority :=  Priority;


// copy command data to header
_cmdHeader := _command;
// call base implementation to copy header to payload buffer
CreateCommandPayload := SUPER^.CreateCommandPayload(AxesGroup := AxesGroup);

// Create logging
CreateCommandPayloadLog(AxesGroup := AxesGroup);
END_METHOD

METHOD INTERNAL CreateCommandPayloadLog
VAR_IN_OUT
  /// Robot assignment of function
  AxesGroup : AxesGroup; 
END_VAR
// Create log entry for Parameter start
CreateLogMessage      ( Timestamp   := AxesGroup.InternalData.SystemTime,
                        MessageType := MessageType.CMD,
                        Severity    := Severity.DEBUG,
                        MessageCode := 0,
                        MessageText := 'Create command payload without additional parameter(s)');
END_METHOD

METHOD FB_init : BOOL
VAR_INPUT
  /// if TRUE, the retain variables are initialized (warm start / cold start)
  bInitRetains : BOOL; 
  /// if TRUE, the instance afterwards gets moved into the copy code (online change)
  bInCopyCode  : BOOL;  
END_VAR
MyType := 'MC_ReadRobotSWLimitsFB';

ExecMode := ExecutionMode.PARALLEL;
END_METHOD

METHOD PROTECTED OnCall
VAR_IN_OUT
  /// Robot assignment of function
  AxesGroup : AxesGroup; 
END_VAR
// call base implementation
SUPER^.OnCall(AxesGroup := AxesGroup);

CASE _stepCmd OF
  
  00:  IF ( _execute_R.Q ) 
       THEN
         // Check function is supported and parameter are valid ?
         IF (( CheckFunctionSupported( AxesGroup := AxesGroup )) AND
             ( CheckParameterValid   ( AxesGroup := AxesGroup )))
         THEN      
           // set busy flag
           Busy := TRUE;
           // Reset command outputs
           SysDepMemSet(pDest := ADR(OutCmd), Value := 0, DataLen := SIZEOF(OutCmd));         
           // apply command parameter
          _parCmd := ParCmd;
           // init parameter sequence
          _command.ParSeq := 1;
           // create command data
           CommandData := CreateCommandPayload(AxesGroup := AxesGroup);
           // Add command to active command register
          _uniqueID := AxesGroup.Acyclic.ActiveCommandRegister.AddCmd( pCommandFB := ADR(THIS^ ));     
           // set timeout
           SetTimeout(PT := _timeoutCmd, rTimer := _timerCmd);
           // inc step counter
          _stepCmd := _stepCmd + 1;
         END_IF 
       END_IF
     

  01:  // Wait for responce received
       IF ( _responseReceived )
       THEN
         // reset response received flag
        _responseReceived := FALSE;

         CASE  _response.State 
         OF
           CmdMessageState.BUFFERED : CommandBuffered := TRUE;
           CmdMessageState.DONE     : Done            := TRUE;
           CmdMessageState.ERROR    : Error           := TRUE;
         END_CASE
                
         // Done, Aborted or Error ?
         IF (_response.State >= CmdMessageState.DONE )
         THEN
           // Reset Busy flag
           Busy := FALSE;
           // Update results
           OutCmd.LimitValues := _response.LimitValues;
           // set timeout
           SetTimeout(PT := _timeoutCmd, rTimer := _timerCmd);
           // inc step counter
          _stepCmd := _stepCmd + 1; 
         END_IF
       END_IF


  02: IF ( NOT Execute)
      THEN
        Reset();
      END_IF     

ELSE
  // invalid step
  ErrorID := RobotLibraryEvents.ERR_INVALID_STEP;
END_CASE


// Reset FB
IF ( NOT Execute )
THEN
  Reset();
END_IF
END_METHOD

METHOD INTERNAL ParseResponsePayload : DINT
VAR_INPUT
  /// Response data
  ResponseData : RobotLibraryRecvDataFB;
  /// Timestamp
  Timestamp    : SystemTime;  
END_VAR
// Table 6-179: Received CMD payload (RC to PLC) of "WriteRobotSWLimits"
// --------------------------
// Header
// --------------------------
// Byte 00 : USINT   - ParSeq | State     
// Byte 01 : SINT    - AlarmMessageSeverity    
// Byte 02 : UINT    - AlarmMessageCode HB
// Byte 03 :         - AlarmMessageCode LB
// --------------------------
// Datablock
// --------------------------
// Byte 04 : IEC_DATE -  Date HW HB;
// Byte 05 :             Date HW LB;
// Byte 06 : IED_TIME -  Time HW HB;
// Byte 07 :             Time HW LB;
// Byte 08 :             Time LW HB;
// Byte 09 :             Time LW LB;
// Byte 10 : REAL        J1LowerLimit HW HB;
// Byte 11 :             J1LowerLimit HW LB;
// Byte 12 :             J1LowerLimit LW HB;
// Byte 13 :             J1LowerLimit LW LB;
// Byte 14 : REAL        J2LowerLimit HW HB;
// Byte 15 :             J2LowerLimit HW LB;
// Byte 16 :             J2LowerLimit LW HB;
// Byte 17 :             J2LowerLimit LW LB;
// Byte 18 : REAL        J3LowerLimit HW HB;
// Byte 19 :             J3LowerLimit HW LB;
// Byte 20 :             J3LowerLimit LW HB;
// Byte 21 :             J3LowerLimit LW LB;
// Byte 22 : REAL        J4LowerLimit HW HB;
// Byte 23 :             J4LowerLimit HW LB;
// Byte 24 :             J4LowerLimit LW HB;
// Byte 25 :             J4LowerLimit LW LB;
// Byte 26 : REAL        J5LowerLimit HW HB;
// Byte 27 :             J5LowerLimit HW LB;
// Byte 28 :             J5LowerLimit LW HB;
// Byte 29 :             J5LowerLimit LW LB;
// Byte 30 : REAL        J6LowerLimit HW HB;
// Byte 31 :             J6LowerLimit HW LB;
// Byte 32 :             J6LowerLimit LW HB;
// Byte 33 :             J6LowerLimit LW LB;
// Byte 34 : REAL        E1LowerLimit HW HB;
// Byte 35 :             E1LowerLimit HW LB;
// Byte 36 :             E1LowerLimit LW HB;
// Byte 37 :             E1LowerLimit LW LB;
// Byte 38 : REAL        J1UpperLimit HW HB;
// Byte 39 :             J1UpperLimit HW LB;
// Byte 40 :             J1UpperLimit LW HB;
// Byte 41 :             J1UpperLimit LW LB;
// Byte 42 : REAL        J2UpperLimit HW HB;
// Byte 43 :             J2UpperLimit HW LB;
// Byte 44 :             J2UpperLimit LW HB;
// Byte 45 :             J2UpperLimit LW LB;
// Byte 46 : REAL        J3UpperLimit HW HB;
// Byte 47 :             J3UpperLimit HW LB;
// Byte 48 :             J3UpperLimit LW HB;
// Byte 49 :             J3UpperLimit LW LB;
// Byte 50 : REAL        J4UpperLimit HW HB;
// Byte 51 :             J4UpperLimit HW LB;
// Byte 52 :             J4UpperLimit LW HB;
// Byte 53 :             J4UpperLimit LW LB;
// Byte 54 : REAL        J5UpperLimit HW HB;
// Byte 55 :             J5UpperLimit HW LB;
// Byte 56 :             J5UpperLimit LW HB;
// Byte 57 :             J5UpperLimit LW LB;
// Byte 58 : REAL        J6UpperLimit HW HB;
// Byte 59 :             J6UpperLimit HW LB;
// Byte 60 :             J6UpperLimit LW HB;
// Byte 61 :             J6UpperLimit LW LB;
// Byte 62 : REAL        E1UpperLimit HW HB;
// Byte 63 :             E1UpperLimit HW LB;
// Byte 64 :             E1UpperLimit LW HB;
// Byte 65 :             E1UpperLimit LW LB;
// Byte 66 : REAL        E2LowerLimit HW HB;
// Byte 67 :             E2LowerLimit HW LB;
// Byte 68 :             E2LowerLimit LW HB;
// Byte 69 :             E2LowerLimit LW LB;
// Byte 70 : REAL        E3LowerLimit HW HB;
// Byte 71 :             E3LowerLimit HW LB;
// Byte 72 :             E3LowerLimit LW HB;
// Byte 73 :             E3LowerLimit LW LB;
// Byte 74 : REAL        E4LowerLimit HW HB;
// Byte 75 :             E4LowerLimit HW LB;
// Byte 76 :             E4LowerLimit LW HB;
// Byte 77 :             E4LowerLimit LW LB;
// Byte 78 : REAL        E5LowerLimit HW HB;
// Byte 79 :             E5LowerLimit HW LB;
// Byte 80 :             E5LowerLimit LW HB;
// Byte 81 :             E5LowerLimit LW LB;
// Byte 82 : REAL        E6LowerLimit HW HB;
// Byte 83 :             E6LowerLimit HW LB;
// Byte 84 :             E6LowerLimit LW HB;
// Byte 85 :             E6LowerLimit LW LB;
// Byte 86 : REAL        E2UpperLimit HW HB;
// Byte 87 :             E2UpperLimit HW LB;
// Byte 88 :             E2UpperLimit LW HB;
// Byte 89 :             E2UpperLimit LW LB;
// Byte 90 : REAL        E3UpperLimit HW HB;
// Byte 91 :             E3UpperLimit HW LB;
// Byte 92 :             E3UpperLimit LW HB;
// Byte 93 :             E3UpperLimit LW LB;
// Byte 94 : REAL        E4UpperLimit HW HB;
// Byte 95 :             E4UpperLimit HW LB;
// Byte 96 :             E4UpperLimit LW HB;
// Byte 97 :             E4UpperLimit LW LB;
// Byte 98 : REAL        E5UpperLimit HW HB;
// Byte 99 :             E5UpperLimit HW LB;
// Byte 100:             E5UpperLimit LW HB;
// Byte 101:             E5UpperLimit LW LB;
// Byte 102: REAL        E6UpperLimit HW HB;
// Byte 103:             E6UpperLimit HW LB;
// Byte 104:             E6UpperLimit LW HB;
// Byte 105:             E6UpperLimit LW LB;
// Byte 106: BOOL        DataChanged;
// --------------------------
// call base implementation to parse the header from payload buffer
ResponseData.PayloadPtr := SUPER^.ParseResponsePayload(ResponseData := ResponseData, Timestamp := Timestamp);

// copy parsed header to response
_response.ParSeq               := _rspHeader.ParSeq;
_response.State                := _rspHeader.State;
_response.AlarmMessageSeverity := _rspHeader.AlarmMessageSeverity;
_response.AlarmMessageCode     := _rspHeader.AlarmMessageCode;

// Get Response.LimitValues.Timestamp.IEC_DATE
_response.LimitValues.Timestamp.IEC_DATE := ResponseData.GetIecDate();
// Get Response.LimitValues.Timestamp.IEC_TIME
_response.LimitValues.Timestamp.IEC_TIME := ResponseData.GetIecTime();
// Get Response.LimitValues.J1LowerLimit
_response.LimitValues.J1LowerLimit := ResponseData.GetReal();
// Get Response.LimitValues.J2LowerLimit
_response.LimitValues.J2LowerLimit := ResponseData.GetReal();
// Get Response.LimitValues.J3LowerLimit
_response.LimitValues.J3LowerLimit := ResponseData.GetReal();
// Get Response.LimitValues.J4LowerLimit
_response.LimitValues.J4LowerLimit := ResponseData.GetReal();
// Get Response.LimitValues.J5LowerLimit
_response.LimitValues.J5LowerLimit := ResponseData.GetReal();
// Get Response.LimitValues.J6LowerLimit
_response.LimitValues.J6LowerLimit := ResponseData.GetReal();
// Get Response.LimitValues.E1LowerLimit
_response.LimitValues.E1LowerLimit := ResponseData.GetReal();
// Get Response.LimitValues.J1UpperLimit
_response.LimitValues.J1UpperLimit := ResponseData.GetReal();
// Get Response.LimitValues.J2UpperLimit
_response.LimitValues.J2UpperLimit := ResponseData.GetReal();
// Get Response.LimitValues.J3UpperLimit
_response.LimitValues.J3UpperLimit := ResponseData.GetReal();
// Get Response.LimitValues.J4UpperLimit
_response.LimitValues.J4UpperLimit := ResponseData.GetReal();
// Get Response.LimitValues.J5UpperLimit
_response.LimitValues.J5UpperLimit := ResponseData.GetReal();
// Get Response.LimitValues.J6UpperLimit
_response.LimitValues.J6UpperLimit := ResponseData.GetReal();
// Get Response.LimitValues.E1UpperLimit
_response.LimitValues.E1UpperLimit := ResponseData.GetReal();
// Get Response.LimitValues.E2LowerLimit
_response.LimitValues.E2LowerLimit := ResponseData.GetReal();
// Get Response.LimitValues.E3LowerLimit
_response.LimitValues.E3LowerLimit := ResponseData.GetReal();
// Get Response.LimitValues.E4LowerLimit
_response.LimitValues.E4LowerLimit := ResponseData.GetReal();
// Get Response.LimitValues.E5LowerLimit
_response.LimitValues.E5LowerLimit := ResponseData.GetReal();
// Get Response.LimitValues.E6LowerLimit
_response.LimitValues.E6LowerLimit := ResponseData.GetReal();
// Get Response.LimitValues.E2UpperLimit
_response.LimitValues.E2UpperLimit := ResponseData.GetReal();
// Get Response.LimitValues.E3UpperLimit
_response.LimitValues.E3UpperLimit := ResponseData.GetReal();
// Get Response.LimitValues.E4UpperLimit
_response.LimitValues.E4UpperLimit := ResponseData.GetReal();
// Get Response.LimitValues.E5UpperLimit
_response.LimitValues.E5UpperLimit := ResponseData.GetReal();
// Get Response.LimitValues.E6UpperLimit
_response.LimitValues.E6UpperLimit := ResponseData.GetReal();

// Create logging
ParseResponsePayloadLog(ResponseData := ResponseData, Timestamp := Timestamp);
END_METHOD

METHOD INTERNAL ParseResponsePayloadLog
VAR_INPUT
  /// Response data
  ResponseData : RobotLibraryRecvDataFB;
  /// Timestamp
  Timestamp    : SystemTime;  
END_VAR
// Create log entry for Parameter start
CreateLogMessage      ( Timestamp   := Timestamp,
                        MessageType := MessageType.CMD,
                        Severity    := Severity.DEBUG,
                        MessageCode := 0,
                        MessageText := 'Parsed the following parameter(s) from response data:');
                        
// Create log entry for LimitValues.Timestamp.IEC_DATE
CreateLogMessagePara1 ( Timestamp   := Timestamp,
                        MessageType := MessageType.CMD,
                        Severity    := Severity.DEBUG,
                        MessageCode := 0,
                        MessageText := 'Response.LimitValues.Timestamp.IEC_DATE = {1}',
                        Para1       :=  IEC_DATE_TO_STRING(_response.LimitValues.Timestamp.IEC_DATE));

// Create log entry for LimitValues.Timestamp.IEC_TIME
CreateLogMessagePara1 ( Timestamp   := Timestamp,
                        MessageType := MessageType.CMD,
                        Severity    := Severity.DEBUG,
                        MessageCode := 0,
                        MessageText := 'Response.LimitValues.Timestamp.IEC_TIME = {1}',
                        Para1       :=  IEC_TIME_TO_STRING(_response.LimitValues.Timestamp.IEC_TIME));
                        
// Create log entry for LimitValues.J1LowerLimit
CreateLogMessagePara1 ( Timestamp   := Timestamp,
                        MessageType := MessageType.CMD,
                        Severity    := Severity.DEBUG,
                        MessageCode := 0,
                        MessageText := 'Response.LimitValues.J1LowerLimit = {1}',
                        Para1       :=  REAL_TO_STRING(_response.LimitValues.J1LowerLimit));

// Create log entry for LimitValues.J2LowerLimit
CreateLogMessagePara1 ( Timestamp   := Timestamp,
                        MessageType := MessageType.CMD,
                        Severity    := Severity.DEBUG,
                        MessageCode := 0,
                        MessageText := 'Response.LimitValues.J2LowerLimit = {1}',
                        Para1       :=  REAL_TO_STRING(_response.LimitValues.J2LowerLimit));

// Create log entry for LimitValues.J3LowerLimit
CreateLogMessagePara1 ( Timestamp   := Timestamp,
                        MessageType := MessageType.CMD,
                        Severity    := Severity.DEBUG,
                        MessageCode := 0,
                        MessageText := 'Response.LimitValues.J3LowerLimit = {1}',
                        Para1       :=  REAL_TO_STRING(_response.LimitValues.J3LowerLimit));

// Create log entry for LimitValues.J4LowerLimit
CreateLogMessagePara1 ( Timestamp   := Timestamp,
                        MessageType := MessageType.CMD,
                        Severity    := Severity.DEBUG,
                        MessageCode := 0,
                        MessageText := 'Response.LimitValues.J4LowerLimit = {1}',
                        Para1       :=  REAL_TO_STRING(_response.LimitValues.J4LowerLimit));

// Create log entry for LimitValues.J5LowerLimit
CreateLogMessagePara1 ( Timestamp   := Timestamp,
                        MessageType := MessageType.CMD,
                        Severity    := Severity.DEBUG,
                        MessageCode := 0,
                        MessageText := 'Response.LimitValues.J5LowerLimit = {1}',
                        Para1       :=  REAL_TO_STRING(_response.LimitValues.J5LowerLimit));

// Create log entry for LimitValues.J6LowerLimit
CreateLogMessagePara1 ( Timestamp   := Timestamp,
                        MessageType := MessageType.CMD,
                        Severity    := Severity.DEBUG,
                        MessageCode := 0,
                        MessageText := 'Response.LimitValues.J6LowerLimit = {1}',
                        Para1       :=  REAL_TO_STRING(_response.LimitValues.J6LowerLimit));

// Create log entry for LimitValues.E1LowerLimit
CreateLogMessagePara1 ( Timestamp   := Timestamp,
                        MessageType := MessageType.CMD,
                        Severity    := Severity.DEBUG,
                        MessageCode := 0,
                        MessageText := 'Response.LimitValues.E1LowerLimit = {1}',
                        Para1       :=  REAL_TO_STRING(_response.LimitValues.E1LowerLimit));

// Create log entry for LimitValues.J1UpperLimit
CreateLogMessagePara1 ( Timestamp   := Timestamp,
                        MessageType := MessageType.CMD,
                        Severity    := Severity.DEBUG,
                        MessageCode := 0,
                        MessageText := 'Response.LimitValues.J1UpperLimit = {1}',
                        Para1       :=  REAL_TO_STRING(_response.LimitValues.J1UpperLimit));

// Create log entry for LimitValues.J2UpperLimit
CreateLogMessagePara1 ( Timestamp   := Timestamp,
                        MessageType := MessageType.CMD,
                        Severity    := Severity.DEBUG,
                        MessageCode := 0,
                        MessageText := 'Response.LimitValues.J2UpperLimit = {1}',
                        Para1       :=  REAL_TO_STRING(_response.LimitValues.J2UpperLimit));

// Create log entry for LimitValues.J3UpperLimit
CreateLogMessagePara1 ( Timestamp   := Timestamp,
                        MessageType := MessageType.CMD,
                        Severity    := Severity.DEBUG,
                        MessageCode := 0,
                        MessageText := 'Response.LimitValues.J3UpperLimit = {1}',
                        Para1       :=  REAL_TO_STRING(_response.LimitValues.J3UpperLimit));

// Create log entry for LimitValues.J4UpperLimit
CreateLogMessagePara1 ( Timestamp   := Timestamp,
                        MessageType := MessageType.CMD,
                        Severity    := Severity.DEBUG,
                        MessageCode := 0,
                        MessageText := 'Response.LimitValues.J4UpperLimit = {1}',
                        Para1       :=  REAL_TO_STRING(_response.LimitValues.J4UpperLimit));

// Create log entry for LimitValues.J5UpperLimit
CreateLogMessagePara1 ( Timestamp   := Timestamp,
                        MessageType := MessageType.CMD,
                        Severity    := Severity.DEBUG,
                        MessageCode := 0,
                        MessageText := 'Response.LimitValues.J5UpperLimit = {1}',
                        Para1       :=  REAL_TO_STRING(_response.LimitValues.J5UpperLimit));

// Create log entry for LimitValues.J6UpperLimit
CreateLogMessagePara1 ( Timestamp   := Timestamp,
                        MessageType := MessageType.CMD,
                        Severity    := Severity.DEBUG,
                        MessageCode := 0,
                        MessageText := 'Response.LimitValues.J6UpperLimit = {1}',
                        Para1       :=  REAL_TO_STRING(_response.LimitValues.J6UpperLimit));

// Create log entry for LimitValues.E1UpperLimit
CreateLogMessagePara1 ( Timestamp   := Timestamp,
                        MessageType := MessageType.CMD,
                        Severity    := Severity.DEBUG,
                        MessageCode := 0,
                        MessageText := 'Response.LimitValues.E1UpperLimit = {1}',
                        Para1       :=  REAL_TO_STRING(_response.LimitValues.E1UpperLimit));

// Create log entry for LimitValues.E2LowerLimit
CreateLogMessagePara1 ( Timestamp   := Timestamp,
                        MessageType := MessageType.CMD,
                        Severity    := Severity.DEBUG,
                        MessageCode := 0,
                        MessageText := 'Response.LimitValues.E2LowerLimit = {1}',
                        Para1       :=  REAL_TO_STRING(_response.LimitValues.E2LowerLimit));

// Create log entry for LimitValues.E3LowerLimit
CreateLogMessagePara1 ( Timestamp   := Timestamp,
                        MessageType := MessageType.CMD,
                        Severity    := Severity.DEBUG,
                        MessageCode := 0,
                        MessageText := 'Response.LimitValues.E3LowerLimit = {1}',
                        Para1       :=  REAL_TO_STRING(_response.LimitValues.E3LowerLimit));

// Create log entry for LimitValues.E4LowerLimit
CreateLogMessagePara1 ( Timestamp   := Timestamp,
                        MessageType := MessageType.CMD,
                        Severity    := Severity.DEBUG,
                        MessageCode := 0,
                        MessageText := 'Response.LimitValues.E4LowerLimit = {1}',
                        Para1       :=  REAL_TO_STRING(_response.LimitValues.E4LowerLimit));

// Create log entry for LimitValues.E5LowerLimit
CreateLogMessagePara1 ( Timestamp   := Timestamp,
                        MessageType := MessageType.CMD,
                        Severity    := Severity.DEBUG,
                        MessageCode := 0,
                        MessageText := 'Response.LimitValues.E5LowerLimit = {1}',
                        Para1       :=  REAL_TO_STRING(_response.LimitValues.E5LowerLimit));

// Create log entry for LimitValues.E6LowerLimit
CreateLogMessagePara1 ( Timestamp   := Timestamp,
                        MessageType := MessageType.CMD,
                        Severity    := Severity.DEBUG,
                        MessageCode := 0,
                        MessageText := 'Response.LimitValues.E6LowerLimit = {1}',
                        Para1       :=  REAL_TO_STRING(_response.LimitValues.E6LowerLimit));

// Create log entry for LimitValues.E2UpperLimit
CreateLogMessagePara1 ( Timestamp   := Timestamp,
                        MessageType := MessageType.CMD,
                        Severity    := Severity.DEBUG,
                        MessageCode := 0,
                        MessageText := 'Response.LimitValues.E2UpperLimit = {1}',
                        Para1       :=  REAL_TO_STRING(_response.LimitValues.E2UpperLimit));

// Create log entry for LimitValues.E3UpperLimit
CreateLogMessagePara1 ( Timestamp   := Timestamp,
                        MessageType := MessageType.CMD,
                        Severity    := Severity.DEBUG,
                        MessageCode := 0,
                        MessageText := 'Response.LimitValues.E3UpperLimit = {1}',
                        Para1       :=  REAL_TO_STRING(_response.LimitValues.E3UpperLimit));

// Create log entry for LimitValues.E4UpperLimit
CreateLogMessagePara1 ( Timestamp   := Timestamp,
                        MessageType := MessageType.CMD,
                        Severity    := Severity.DEBUG,
                        MessageCode := 0,
                        MessageText := 'Response.LimitValues.E4UpperLimit = {1}',
                        Para1       :=  REAL_TO_STRING(_response.LimitValues.E4UpperLimit));

// Create log entry for LimitValues.E5UpperLimit
CreateLogMessagePara1 ( Timestamp   := Timestamp,
                        MessageType := MessageType.CMD,
                        Severity    := Severity.DEBUG,
                        MessageCode := 0,
                        MessageText := 'Response.LimitValues.E5UpperLimit = {1}',
                        Para1       :=  REAL_TO_STRING(_response.LimitValues.E5UpperLimit));

// Create log entry for LimitValues.E6UpperLimit
CreateLogMessagePara1 ( Timestamp   := Timestamp,
                        MessageType := MessageType.CMD,
                        Severity    := Severity.DEBUG,
                        MessageCode := 0,
                        MessageText := 'Response.LimitValues.E6UpperLimit = {1}',
                        Para1       :=  REAL_TO_STRING(_response.LimitValues.E6UpperLimit));
END_METHOD

METHOD PROTECTED Reset : DINT
VAR_INPUT
END_VAR
Reset := SUPER^.Reset();

Done               := FALSE;
Busy               := FALSE;
CommandBuffered    := FALSE;
END_METHOD

END_FUNCTION_BLOCK

// Library/POUs/Read/MC_ReadSystemVariable/MC_ReadSystemVariableFB
/// Read specific parameter of the robot
FUNCTION_BLOCK MC_ReadSystemVariableFB EXTENDS RobotLibraryBaseExecuteFB
// ------------------------------------------------------------------------- 
//  SRCI Robot Library                                                
// ------------------------------------------------------------------------- 
//                                                                           
//  Object:      ReadSystemVariableFB                                       
//  Author:      Thorsten Brach                                                
//  Date:        2024-06-01
//
//  Description:                                              
//   
//                                                                           
//  Copyright: 
//    (C) 2024 Thorsten Brach. All rights reserved                                                                                                                                            
//             Licensed under the LGPL-3.0 license.
//                                                                           
//  Disclaimer:                                                                           
//    This project is provided without any guarantee and can be used for   
//    private and commercial purposes. Any use is at the user’s 
//    own risk and responsibility.
//
// -------------------------------------------------------------------------
VAR_INPUT
  /// Processing Mode
  ProcessingMode     : ProcessingMode;
  /// Defines the target sequence in which the command will be executed
  SequenceFlag       : SequenceFlag;
  /// command parameter 
  ParCmd             : ReadSystemVariableParCmd;
END_VAR
VAR_OUTPUT
  /// TRUE, while the following outputs return valid values:
  /// • DataType
  /// • Data_0
  /// • Data_1
  /// • Data_2
  /// • Data_3
  /// • Data_4
  /// • Data_5
  /// • Data_6
  /// • Data_7
  Valid              : BOOL; 
  /// Command is transferred and confirmed by the RC
  CommandBuffered    : BOOL;
  /// The command was aborted by another command.
  CommandAborted     : BOOL;
  /// TRUE, while command is interrupted during execution and can be continued
  CommandInterrupted : BOOL;
  /// Receiving of input parameter values has been acknowledged by RC
  ParameterAccepted  : BOOL;
  /// command outputs
  OutCmd             : ReadSystemVariableOutCmd;       
END_VAR

VAR
  /// internal copy of command parameter 
 _parCmd             : ReadSystemVariableParCmd;
  /// command data to send
 _command            : ReadSystemVariableSendData;
  /// response data received
 _response           : ReadSystemVariableRecvData;      
END_VAR

SUPER^(AxesGroup := AxesGroup);

METHOD PROTECTED CheckFunctionSupported : BOOL
VAR_IN_OUT
  /// Robot assignment of function
  AxesGroup : AxesGroup; 
END_VAR
CheckFunctionSupported := AxesGroup.InternalData.RCSupportedFunctions.ReadSystemVariable;

IF ( NOT CheckFunctionSupported )
THEN
  // call base implementation for set error and create log entry
  SUPER^.CheckFunctionSupported(AxesGroup := AxesGroup);
END_IF
END_METHOD

METHOD PROTECTED CheckParameterChanged : BOOL
VAR_IN_OUT
  /// Robot assignment of function
  AxesGroup    : AxesGroup; 
END_VAR
// Check ParCmd Size is > 0, because MemCmp does not work correctly with size = 0
IF (SIZEOF(ParCmd) = 0) 
THEN 
  RETURN;
END_IF

// compare memory 
_parameterChanged := ( SysDepMemCmp(pData1 := ADR(ParCmd), pData2 := ADR(_parCmd), DataLen := SIZEOF(ParCmd)) <> RobotLibraryConstants.OK );

// check parameter valid ?
_parameterValid   := CheckParameterValid( AxesGroup := AxesGroup );

IF ((  _parameterChanged        )  AND 
    (  _parameterValid          )) OR
    (  _parameterUpdateInternal )  
THEN  
  // reset internal flag for send parameter update
 _parameterUpdateInternal := FALSE;
  // update internal copy of parameters 
 _parCmd := ParCmd;
  // inc parameter sequence
 _command.ParSeq := _command.ParSeq + 1;
  // update command data  
  CommandData := CreateCommandPayload(AxesGroup := AxesGroup); // ( Access via reference to rCommandFB in ACR )
  // notify active command register 
  AxesGroup.Acyclic.ActiveCommandRegister.NotifyParameterChanged := _uniqueID;
  // Reset parameter accepted flag
  ParameterAccepted := FALSE;  
END_IF
END_METHOD

METHOD INTERNAL CreateCommandPayload : RobotLibrarySendDataFB
VAR_IN_OUT
  /// Robot assignment of function
  AxesGroup : AxesGroup; 
END_VAR
// Table 6-618: Sent CMD payload (PLC to RC) of "ReadSystemVariable"
// --------------------------
// Header
// --------------------------
// Byte 00 : UINT  - Type HB     
// Byte 01 :       - Type LB    
// Byte 02 : USINT - Reserve | ExecutionMode
// Byte 03 : USINT - ParSeq  | Priority
// --------------------------
// Datablock
// --------------------------
// Byte 04 : SINT  EmitterID[0];
// Byte 05 : SINT  EmitterID[1];
// Byte 06 : SINT  EmitterID[2];
// Byte 07 : SINT  EmitterID[3];
// Byte 08 : SINT  ListenerID;
// Byte 09 : BYTE  Reserved;
// Byte 10 : UINT  ParameterID[0] HW HB;
// Byte 11 :       ParameterID[0] HW LB;
// Byte 12 : UINT  ParameterID[1] HW HB;
// Byte 13 :       ParameterID[1] HW LB;
// Byte 14 : UINT  ParameterID[2] HW HB;
// Byte 15 :       ParameterID[2] HW LB;
// Byte 16 : UINT  ParameterID[3] HW HB;
// Byte 17 :       ParameterID[3] HW LB;
// Byte 18 : UINT  ParameterID[4] HW HB;
// Byte 19 :       ParameterID[4] HW LB;
// Byte 20 : UINT  ParameterID[5] HW HB;
// Byte 21 :       ParameterID[5] HW LB;
// Byte 22 : UINT  ParameterID[6] HW HB;
// Byte 23 :       ParameterID[6] HW LB;
// Byte 24 : UINT  ParameterID[7] HW HB;
// Byte 25 :       ParameterID[7] HW LB;
// Byte 26 : USINT SubParameterID[0];
// Byte 27 : USINT SubParameterID[1];
// Byte 28 : USINT SubParameterID[2];
// Byte 29 : USINT SubParameterID[3];
// Byte 30 : USINT SubParameterID[4];
// Byte 31 : USINT SubParameterID[5];
// Byte 32 : USINT SubParameterID[6];
// Byte 33 : USINT SubParameterID[7];
// Byte 34 : BOOL  RCParameter;

// --------------------------
VAR
  /// internal index for loops
 _idx : DINT;
END_VAR
// set command parameter 
_command.CmdTyp         :=  CmdType.ReadSystemVariable;
_command.ExecMode       :=  ExecMode;
_command.ParSeq         := _command.ParSeq;
_command.Priority       :=  Priority;
_command.EmitterID[0]   := 0;
_command.EmitterID[1]   := 0;
_command.EmitterID[2]   := 0;
_command.EmitterID[3]   := 0;
_command.Reserve        := 0;
_command.ListenerID     := _parCmd.ListenerID;
_command.ParameterID    := _parCmd.ParameterID;
_command.SubParameterID := _parCmd.SubParameterID;
_command.RCParameter    := _parCmd.RCParameter;


// copy command data to header
_cmdHeader := _command;
// call base implementation to copy header to payload buffer
CreateCommandPayload := SUPER^.CreateCommandPayload(AxesGroup := AxesGroup);

// add command.EmitterID[0]
CreateCommandPayload.AddSint(_command.EmitterID[0]);
// add command.EmitterID[1]
CreateCommandPayload.AddSint(_command.EmitterID[1]);
// add command.EmitterID[2]
CreateCommandPayload.AddSint(_command.EmitterID[2]);
// add command.EmitterID[3]
CreateCommandPayload.AddSint(_command.EmitterID[3]);
// add command.ListenerID
CreateCommandPayload.AddSint(_command.ListenerID);
// add command.Reserve
CreateCommandPayload.AddByte(_command.Reserve);

FOR _idx := 0 TO 7 
DO
  // add command.ParameterID[_idx]
  CreateCommandPayload.AddUint(_command.ParameterID[_idx]);
END_FOR

FOR _idx := 0 TO 7 
DO
  // add command.SubParameterID[_idx]
  CreateCommandPayload.AddUsint(_command.SubParameterID[_idx]);
END_FOR

// add command.RCParameter
CreateCommandPayload.AddBool(_command.RCParameter);

// Create logging
CreateCommandPayloadLog(AxesGroup := AxesGroup);
END_METHOD

METHOD INTERNAL CreateCommandPayloadLog
VAR_IN_OUT
  /// Robot assignment of function
  AxesGroup : AxesGroup; 
END_VAR
VAR 
  /// internal index for loops
 _idx : DINT;
END_VAR
// Create log entry for Parameter start
CreateLogMessage      ( Timestamp   := AxesGroup.InternalData.SystemTime,
                        MessageType := MessageType.CMD,
                        Severity    := Severity.DEBUG,
                        MessageCode := 0,
                        MessageText := 'Create command payload with the following parameter(s) :');
  
// Create log entry for EmitterID[x]
FOR _idx := 0 TO 3
DO
  CreateLogMessagePara2 ( Timestamp   := AxesGroup.InternalData.SystemTime,
                          MessageType := MessageType.CMD,
                          Severity    := Severity.DEBUG,
                          MessageCode := 0,
                          MessageText := 'Command.EmitterID[{2}] = {1}',
                          Para1       :=  SINT_TO_STRING(_command.EmitterID[_idx]),
                          Para2       :=  DINT_TO_STRING(_idx));
END_FOR

// Create log entry for ListenerID
CreateLogMessagePara1 ( Timestamp   := AxesGroup.InternalData.SystemTime,
                        MessageType := MessageType.CMD,
                        Severity    := Severity.DEBUG,
                        MessageCode := 0,
                        MessageText := 'Command.ListenerID = {1}',
                        Para1       :=  SINT_TO_STRING(_command.ListenerID));
                        
// Create log entry for Reserve
CreateLogMessagePara1 ( Timestamp   := AxesGroup.InternalData.SystemTime,
                        MessageType := MessageType.CMD,
                        Severity    := Severity.DEBUG,
                        MessageCode := 0,
                        MessageText := 'Command.Reserve = {1}',
                        Para1       :=  BYTE_TO_STRING(_command.Reserve));

// Create log entry for ParameterID[x]
FOR _idx := 0 TO 7
DO
  CreateLogMessagePara2 ( Timestamp   := AxesGroup.InternalData.SystemTime,
                          MessageType := MessageType.CMD,
                          Severity    := Severity.DEBUG,
                          MessageCode := 0,
                          MessageText := 'Command.ParameterID[{2}] = {1}',
                          Para1       :=  UINT_TO_STRING(_command.ParameterID[_idx]),
                          Para2       :=  DINT_TO_STRING(_idx));
END_FOR

// Create log entry for SubParameterID[x]
FOR _idx := 0 TO 7
DO
  CreateLogMessagePara2 ( Timestamp   := AxesGroup.InternalData.SystemTime,
                          MessageType := MessageType.CMD,
                          Severity    := Severity.DEBUG,
                          MessageCode := 0,
                          MessageText := 'Command.SubParameterID[{2}] = {1}',
                          Para1       :=  USINT_TO_STRING(_command.SubParameterID[_idx]),
                          Para2       :=  DINT_TO_STRING(_idx));
END_FOR


// Create log entry for RCParameter
CreateLogMessagePara1 ( Timestamp   := AxesGroup.InternalData.SystemTime,
                        MessageType := MessageType.CMD,
                        Severity    := Severity.DEBUG,
                        MessageCode := 0,
                        MessageText := 'Command.RCParameter = {1}',
                        Para1       :=  BOOL_TO_STRING(_command.RCParameter));
END_METHOD

METHOD FB_init : BOOL
VAR_INPUT
  /// if TRUE, the retain variables are initialized (warm start / cold start)
  bInitRetains : BOOL; 
  /// if TRUE, the instance afterwards gets moved into the copy code (online change)
  bInCopyCode  : BOOL;  
END_VAR
MyType := 'MC_ReadSystemVariableFB';

ExecMode := ExecutionMode.PARALLEL;
END_METHOD

METHOD PROTECTED OnCall
VAR_IN_OUT
  /// Robot assignment of function
  AxesGroup : AxesGroup; 
END_VAR
// call base implementation
SUPER^.OnCall(AxesGroup := AxesGroup);

CASE _stepCmd OF
  
  00:  IF ( _execute_R.Q )  
       THEN
         // Check function is supported and parameter are valid ?
         IF (( CheckFunctionSupported( AxesGroup := AxesGroup )) AND
             ( CheckParameterValid   ( AxesGroup := AxesGroup )))
         THEN      
           // set busy flag
           Busy := TRUE;
           // Reset command outputs
           SysDepMemSet(pDest := ADR(OutCmd), Value := 0, DataLen := SIZEOF(OutCmd));         
           // apply command parameter
          _parCmd := ParCmd;
           // init parameter sequence
          _command.ParSeq := 1;
           // create command data
           CommandData := CreateCommandPayload(AxesGroup := AxesGroup);
           // Add command to active command register
          _uniqueID := AxesGroup.Acyclic.ActiveCommandRegister.AddCmd( pCommandFB := ADR(THIS^ ));     
           // set timeout
           SetTimeout(PT := _timeoutCmd, rTimer := _timerCmd);
           // inc step counter
          _stepCmd := _stepCmd + 1;
         END_IF 
       END_IF
     

  01:  // Wait for responce received
       IF ( _responseReceived )
       THEN
         // reset response received flag
        _responseReceived := FALSE;

         CASE  _response.State 
         OF
           CmdMessageState.BUFFERED    : CommandBuffered    := TRUE;
           CmdMessageState.ACTIVE      : ParameterAccepted  := TRUE;
           CmdMessageState.INTERRUPTED : CommandInterrupted := TRUE;           
           CmdMessageState.DONE        : Done               := TRUE;
           CmdMessageState.ABORTED     : CommandAborted     := TRUE;
           CmdMessageState.ERROR       : Error              := TRUE;
         END_CASE
                
         // Done, Aborted or Error ?
         IF (_response.State >= CmdMessageState.DONE )
         THEN
           // Reset Busy flag
           Busy := FALSE;
           // Update results
           OutCmd.OriginID          := _response.OriginID;
           OutCmd.InvocationCounter := _response.InvocationCounter;
           OutCmd.DataType          := _response.DataType;
           OutCmd.Data_0            := _response.Data_0;
           OutCmd.Data_1            := _response.Data_1;
           OutCmd.Data_2            := _response.Data_2;
           OutCmd.Data_3            := _response.Data_3;
           OutCmd.Data_4            := _response.Data_4;
           OutCmd.Data_5            := _response.Data_5;
           OutCmd.Data_6            := _response.Data_6;
           OutCmd.Data_7            := _response.Data_7;
           
           // set timeout
           SetTimeout(PT := _timeoutCmd, rTimer := _timerCmd);
           // inc step counter
          _stepCmd := _stepCmd + 1; 
         END_IF
       END_IF


  02: IF ( NOT Execute)
      THEN
        Reset();
      END_IF     

ELSE
  // invalid step
  ErrorID := RobotLibraryEvents.ERR_INVALID_STEP;
END_CASE


// Reset FB
IF ( NOT Execute )
THEN
  Reset();
END_IF
END_METHOD

